LIN {X 0,Y 449.895,Z 770.969,A -85,B 0,C 180,E1 -4613.165,E2 -4613.165} C_VEL
LIN {X 0,Y 451.158,Z 755.212,A -85,B 0,C 180,E1 -4614.344,E2 -4614.344} C_VEL
LIN {X 0,Y 452.253,Z 738.74,A -85,B 0,C 180,E1 -4615.328,E2 -4615.328} C_VEL
LIN {X 0,Y 453.129,Z 720.861,A -85,B 0,C 180,E1 -4616.147,E2 -4616.147} C_VEL
LIN {X 0,Y 453.677,Z 702.427,A -85,B 0,C 180,E1 -4616.749,E2 -4616.749} C_VEL
LIN {X 0,Y 453.972,Z 680.153,A -85,B 0,C 180,E1 -4617.195,E2 -4617.195} C_VEL
LIN {X 0,Y 457.144,Z 495.027,A -85,B 0,C 180,E1 -4620.269,E2 -4620.269} C_VEL
LIN {X 0,Y 456.167,Z 488.518,A -85,B 0,C 180,E1 -4620.474,E2 -4620.474} C_VEL
LIN {X 0,Y 456.984,Z 456.622,A -85,B 0,C 180,E1 -4622.788,E2 -4622.788} C_VEL
LIN {X 0,Y 458.772,Z 418.991,A -85,B 0,C 180,E1 -4625.739,E2 -4625.739} C_VEL
LIN {X 0,Y 451.224,Z 399.096,A -85,B 0,C 180,E1 -4628.127,E2 -4628.127} C_VEL
LIN {X 0,Y 444.43,Z 383.394,A -85,B 0,C 180,E1 -4630.1,E2 -4630.1} C_VEL
LIN {X 0,Y 441.262,Z 376.238,A -85,B 0,C 180,E1 -4631.014,E2 -4631.014} C_VEL
LIN {X 0,Y 441.194,Z 375.762,A -85,B 0,C 180,E1 -4631.088,E2 -4631.088} C_VEL
LIN {X 0,Y 441.156,Z 375.762,A -85,B 0,C 180,E1 -4634.819,E2 -4634.819} C_VEL
LIN {X 0,Y 441.18,Z 375.869,A -85,B 0,C 180,E1 -4634.958,E2 -4634.958} C_VEL
LIN {X 0,Y 442.687,Z 379.535,A -85,B 0,C 180,E1 -4635.559,E2 -4635.559} C_VEL
LIN {X 0,Y 450.981,Z 398.056,A -85,B 0,C 180,E1 -4638.537,E2 -4638.537} C_VEL
LIN {X 0,Y 459.04,Z 417.845,A -85,B 0,C 180,E1 -4641.441,E2 -4641.441} C_VEL
LIN {X 0,Y 461.711,Z 425.418,A -85,B 0,C 180,E1 -4642.476,E2 -4642.476} C_VEL
LIN {X 0,Y 458.465,Z 467.127,A -85,B 0,C 180,E1 -4646.211,E2 -4646.211} C_VEL
LIN {X 0,Y 455.403,Z 509.659,A -85,B 0,C 180,E1 -4649.961,E2 -4649.961} C_VEL
LIN {X 0,Y 452.531,Z 553.564,A -85,B 0,C 180,E1 -4653.775,E2 -4653.775} C_VEL
LIN {X 0,Y 449.914,Z 598.968,A -85,B 0,C 180,E1 -4657.665,E2 -4657.665} C_VEL
LIN {X 0,Y 450.757,Z 607.685,A -85,B 0,C 180,E1 -4657.915,E2 -4657.915} C_VEL
LIN {X 0,Y 447.26,Z 745.636,A -85,B 0,C 180,E1 -4660.73,E2 -4660.73} C_VEL
LIN {X 0,Y 446.843,Z 762.879,A -85,B 0,C 180,E1 -4661.338,E2 -4661.338} C_VEL
LIN {X 0,Y 446.246,Z 778.27,A -85,B 0,C 180,E1 -4662.123,E2 -4662.123} C_VEL
LIN {X 0,Y 445.489,Z 793.673,A -85,B 0,C 180,E1 -4663.17,E2 -4663.17} C_VEL
LIN {X 0,Y 444.687,Z 807.201,A -85,B 0,C 180,E1 -4664.346,E2 -4664.346} C_VEL
LIN {X 0,Y 443.839,Z 820.409,A -85,B 0,C 180,E1 -4665.785,E2 -4665.785} C_VEL
LIN {X 0,Y 443.061,Z 831.979,A -85,B 0,C 180,E1 -4667.355,E2 -4667.355} C_VEL
LIN {X 0,Y 442.35,Z 842.758,A -85,B 0,C 180,E1 -4669.186,E2 -4669.186} C_VEL
LIN {X 0,Y 441.823,Z 851.245,A -85,B 0,C 180,E1 -4671.016,E2 -4671.016} C_VEL
LIN {X 0,Y 441.424,Z 858.712,A -85,B 0,C 180,E1 -4673.105,E2 -4673.105} C_VEL
LIN {X 0,Y 441.19,Z 863.794,A -85,B 0,C 180,E1 -4675.059,E2 -4675.059} C_VEL
LIN {X 0,Y 441.097,Z 867.62,A -85,B 0,C 180,E1 -4677.271,E2 -4677.271} C_VEL
LIN {X 0,Y 441.088,Z 869.436,A -85,B 0,C 180,E1 -4679.35,E2 -4679.35} C_VEL
LIN {X 0,Y 441.194,Z 869.55,A -85,B 0,C 180,E1 -4681.558,E2 -4681.558} C_VEL
LIN {X 0,Y 441.366,Z 867.927,A -85,B 0,C 180,E1 -4683.636,E2 -4683.636} C_VEL
LIN {X 0,Y 441.715,Z 864.344,A -85,B 0,C 180,E1 -4685.846,E2 -4685.846} C_VEL
LIN {X 0,Y 442.16,Z 859.396,A -85,B 0,C 180,E1 -4687.797,E2 -4687.797} C_VEL
LIN {X 0,Y 442.811,Z 852.654,A -85,B 0,C 180,E1 -4689.75,E2 -4689.75} C_VEL
LIN {X 0,Y 443.571,Z 844.422,A -85,B 0,C 180,E1 -4691.573,E2 -4691.573} C_VEL
LIN {X 0,Y 444.542,Z 833.949,A -85,B 0,C 180,E1 -4693.395,E2 -4693.395} C_VEL
LIN {X 0,Y 445.533,Z 822.497,A -85,B 0,C 180,E1 -4694.956,E2 -4694.956} C_VEL
LIN {X 0,Y 446.52,Z 810.059,A -85,B 0,C 180,E1 -4696.321,E2 -4696.321} C_VEL
LIN {X 0,Y 447.465,Z 795.723,A -85,B 0,C 180,E1 -4697.557,E2 -4697.557} C_VEL
LIN {X 0,Y 448.16,Z 782.092,A -85,B 0,C 180,E1 -4698.47,E2 -4698.47} C_VEL
LIN {X 0,Y 448.749,Z 765.732,A -85,B 0,C 180,E1 -4699.288,E2 -4699.288} C_VEL
LIN {X 0,Y 449.106,Z 747.084,A -85,B 0,C 180,E1 -4699.911,E2 -4699.911} C_VEL
LIN {X 0,Y 452.046,Z 696.665,A -85,B 0,C 180,E1 -4701.377,E2 -4701.377} C_VEL
LIN {X 0,Y 458.354,Z 622.755,A -85,B 0,C 180,E1 -4703.596,E2 -4703.596} C_VEL
LIN {X 0,Y 461.651,Z 613.359,A -85,B 0,C 180,E1 -4704.241,E2 -4704.241} C_VEL
LIN {X 0,Y 468.36,Z 575.653,A -85,B 0,C 180,E1 -4708.081,E2 -4708.081} C_VEL
LIN {X 0,Y 475.645,Z 546.296,A -85,B 0,C 180,E1 -4711.28,E2 -4711.28} C_VEL
LIN {X 0,Y 482.867,Z 525.512,A -85,B 0,C 180,E1 -4713.706,E2 -4713.706} C_VEL
LIN {X 0,Y 490.96,Z 508.824,A -85,B 0,C 180,E1 -4715.802,E2 -4715.802} C_VEL
LIN {X 0,Y 485.466,Z 518.576,A -85,B 0,C 180,E1 -4717.344,E2 -4717.344} C_VEL
LIN {X 0,Y 482.77,Z 527.164,A -85,B 0,C 180,E1 -4718.716,E2 -4718.716} C_VEL
LIN {X 0,Y 482.118,Z 536.127,A -85,B 0,C 180,E1 -4720.164,E2 -4720.164} C_VEL
LIN {X 0,Y 483.586,Z 544.905,A -85,B 0,C 180,E1 -4721.582,E2 -4721.582} C_VEL
LIN {X 0,Y 487.497,Z 554.414,A -85,B 0,C 180,E1 -4723.1,E2 -4723.1} C_VEL
LIN {X 0,Y 493.464,Z 563.318,A -85,B 0,C 180,E1 -4724.512,E2 -4724.512} C_VEL
LIN {X 0,Y 501.507,Z 571.927,A -85,B 0,C 180,E1 -4725.867,E2 -4725.867} C_VEL
LIN {X 0,Y 512.262,Z 580.404,A -85,B 0,C 180,E1 -4727.214,E2 -4727.214} C_VEL
LIN {X 0,Y 520.948,Z 586.006,A -85,B 0,C 180,E1 -4728.093,E2 -4728.093} C_VEL
LIN {X 0,Y 500.898,Z 618.864,A -85,B 0,C 180,E1 -4728.811,E2 -4728.811} C_VEL
LIN {X 0,Y 489.956,Z 639.653,A -85,B 0,C 180,E1 -4729.388,E2 -4729.388} C_VEL
LIN {X 0,Y 482.648,Z 656.795,A -85,B 0,C 180,E1 -4729.989,E2 -4729.989} C_VEL
LIN {X 0,Y 479.917,Z 663.519,A -85,B 0,C 180,E1 -4730.237,E2 -4730.237} C_VEL
LIN {X 0,Y 472.657,Z 680.377,A -85,B 0,C 180,E1 -4730.843,E2 -4730.843} C_VEL
LIN {X 0,Y 463.801,Z 707.381,A -85,B 0,C 180,E1 -4732.013,E2 -4732.013} C_VEL
LIN {X 0,Y 462.854,Z 711.533,A -85,B 0,C 180,E1 -4732.171,E2 -4732.171} C_VEL
LIN {X 0,Y 461.732,Z 725.369,A -85,B 0,C 180,E1 -4732.362,E2 -4732.362} C_VEL
LIN {X 0,Y 460.813,Z 757.516,A -85,B 0,C 180,E1 -4732.978,E2 -4732.978} C_VEL
LIN {X 0,Y 459.501,Z 781.218,A -85,B 0,C 180,E1 -4733.648,E2 -4733.648} C_VEL
LIN {X 0,Y 457.971,Z 803.987,A -85,B 0,C 180,E1 -4734.522,E2 -4734.522} C_VEL
LIN {X 0,Y 456.223,Z 826.917,A -85,B 0,C 180,E1 -4735.643,E2 -4735.643} C_VEL
LIN {X 0,Y 454.282,Z 849.228,A -85,B 0,C 180,E1 -4736.988,E2 -4736.988} C_VEL
LIN {X 0,Y 452.395,Z 869.681,A -85,B 0,C 180,E1 -4738.486,E2 -4738.486} C_VEL
LIN {X 0,Y 450.357,Z 889.784,A -85,B 0,C 180,E1 -4740.235,E2 -4740.235} C_VEL
LIN {X 0,Y 448.559,Z 907.091,A -85,B 0,C 180,E1 -4741.998,E2 -4741.998} C_VEL
LIN {X 0,Y 446.629,Z 925.029,A -85,B 0,C 180,E1 -4744.151,E2 -4744.151} C_VEL
LIN {X 0,Y 444.866,Z 941.503,A -85,B 0,C 180,E1 -4746.49,E2 -4746.49} C_VEL
LIN {X 0,Y 443.317,Z 956.495,A -85,B 0,C 180,E1 -4749.024,E2 -4749.024} C_VEL
LIN {X 0,Y 442.11,Z 968.957,A -85,B 0,C 180,E1 -4751.541,E2 -4751.541} C_VEL
LIN {X 0,Y 441.355,Z 977.773,A -85,B 0,C 180,E1 -4753.685,E2 -4753.685} C_VEL
LIN {X 0,Y 440.635,Z 986.687,A -85,B 0,C 180,E1 -4756.483,E2 -4756.483} C_VEL
LIN {X 0,Y 440.219,Z 993.705,A -85,B 0,C 180,E1 -4759.266,E2 -4759.266} C_VEL
LIN {X 0,Y 440.005,Z 999.024,A -85,B 0,C 180,E1 -4762.032,E2 -4762.032} C_VEL
LIN {X 0,Y 439.912,Z 1002.741,A -85,B 0,C 180,E1 -4764.783,E2 -4764.783} C_VEL
LIN {X 0,Y 439.9,Z 1004.828,A -85,B 0,C 180,E1 -4767.525,E2 -4767.525} C_VEL
LIN {X 0,Y 439.894,Z 1005.447,A -85,B 0,C 180,E1 -4770.521,E2 -4770.521} C_VEL
LIN {X 0,Y 439.906,Z 1004.417,A -85,B 0,C 180,E1 -4773.257,E2 -4773.257} C_VEL
LIN {X 0,Y 439.948,Z 1001.676,A -85,B 0,C 180,E1 -4776.131,E2 -4776.131} C_VEL
LIN {X 0,Y 440.067,Z 997.197,A -85,B 0,C 180,E1 -4779.019,E2 -4779.019} C_VEL
LIN {X 0,Y 440.339,Z 991.238,A -85,B 0,C 180,E1 -4781.792,E2 -4781.792} C_VEL
LIN {X 0,Y 440.857,Z 983.531,A -85,B 0,C 180,E1 -4784.581,E2 -4784.581} C_VEL
LIN {X 0,Y 441.556,Z 975.224,A -85,B 0,C 180,E1 -4786.984,E2 -4786.984} C_VEL
LIN {X 0,Y 442.585,Z 964.124,A -85,B 0,C 180,E1 -4789.533,E2 -4789.533} C_VEL
LIN {X 0,Y 443.881,Z 951.647,A -85,B 0,C 180,E1 -4791.957,E2 -4791.957} C_VEL
LIN {X 0,Y 445.543,Z 936.945,A -85,B 0,C 180,E1 -4794.388,E2 -4794.388} C_VEL
LIN {X 0,Y 447.541,Z 920.085,A -85,B 0,C 180,E1 -4796.755,E2 -4796.755} C_VEL
LIN {X 0,Y 449.799,Z 901.306,A -85,B 0,C 180,E1 -4798.985,E2 -4798.985} C_VEL
LIN {X 0,Y 452.216,Z 881.067,A -85,B 0,C 180,E1 -4801.008,E2 -4801.008} C_VEL
LIN {X 0,Y 454.533,Z 861.152,A -85,B 0,C 180,E1 -4802.686,E2 -4802.686} C_VEL
LIN {X 0,Y 456.76,Z 840.526,A -85,B 0,C 180,E1 -4804.132,E2 -4804.132} C_VEL
LIN {X 0,Y 458.846,Z 819.523,A -85,B 0,C 180,E1 -4805.348,E2 -4805.348} C_VEL
LIN {X 0,Y 460.789,Z 797.618,A -85,B 0,C 180,E1 -4806.368,E2 -4806.368} C_VEL
LIN {X 0,Y 462.401,Z 775.254,A -85,B 0,C 180,E1 -4807.157,E2 -4807.157} C_VEL
LIN {X 0,Y 463.714,Z 752.034,A -85,B 0,C 180,E1 -4807.736,E2 -4807.736} C_VEL
LIN {X 0,Y 464.958,Z 716.912,A -85,B 0,C 180,E1 -4808.352,E2 -4808.352} C_VEL
LIN {X 0,Y 465.536,Z 714.104,A -85,B 0,C 180,E1 -4808.446,E2 -4808.446} C_VEL
LIN {X 0,Y 470.715,Z 697.809,A -85,B 0,C 180,E1 -4809.192,E2 -4809.192} C_VEL
LIN {X 0,Y 477.201,Z 679.573,A -85,B 0,C 180,E1 -4809.955,E2 -4809.955} C_VEL
LIN {X 0,Y 485.1,Z 661.285,A -85,B 0,C 180,E1 -4810.563,E2 -4810.563} C_VEL
LIN {X 0,Y 492.217,Z 644.342,A -85,B 0,C 180,E1 -4811.159,E2 -4811.159} C_VEL
LIN {X 0,Y 502.709,Z 623.858,A -85,B 0,C 180,E1 -4811.705,E2 -4811.705} C_VEL
LIN {X 0,Y 519.668,Z 594.789,A -85,B 0,C 180,E1 -4812.256,E2 -4812.256} C_VEL
LIN {X 0,Y 523.657,Z 588.098,A -85,B 0,C 180,E1 -4812.36,E2 -4812.36} C_VEL
LIN {X 0,Y 513.143,Z 581.511,A -85,B 0,C 180,E1 -4813.707,E2 -4813.707} C_VEL
LIN {X 0,Y 503.509,Z 573.197,A -85,B 0,C 180,E1 -4815.175,E2 -4815.175} C_VEL
LIN {X 0,Y 495.035,Z 562.874,A -85,B 0,C 180,E1 -4816.788,E2 -4816.788} C_VEL
LIN {X 0,Y 488.639,Z 551.749,A -85,B 0,C 180,E1 -4818.319,E2 -4818.319} C_VEL
LIN {X 0,Y 483.581,Z 538.76,A -85,B 0,C 180,E1 -4819.908,E2 -4819.908} C_VEL
LIN {X 0,Y 480.199,Z 523.859,A -85,B 0,C 180,E1 -4821.526,E2 -4821.526} C_VEL
LIN {X 0,Y 478.615,Z 506.943,A -85,B 0,C 180,E1 -4823.162,E2 -4823.162} C_VEL
LIN {X 0,Y 478.809,Z 488.569,A -85,B 0,C 180,E1 -4824.735,E2 -4824.735} C_VEL
LIN {X 0,Y 482.727,Z 450.056,A -85,B 0,C 180,E1 -4827.698,E2 -4827.698} C_VEL
LIN {X 0,Y 473.244,Z 432.509,A -85,B 0,C 180,E1 -4830.788,E2 -4830.788} C_VEL
LIN {X 0,Y 465.807,Z 419.157,A -85,B 0,C 180,E1 -4833.345,E2 -4833.345} C_VEL
LIN {X 0,Y 458.025,Z 405.408,A -85,B 0,C 180,E1 -4836.181,E2 -4836.181} C_VEL
LIN {X 0,Y 452.378,Z 395.654,A -85,B 0,C 180,E1 -4838.34,E2 -4838.34} C_VEL
LIN {X 0,Y 449.617,Z 390.88,A -85,B 0,C 180,E1 -4839.43,E2 -4839.43} C_VEL
LIN {X 0,Y 447.276,Z 386.724,A -85,B 0,C 180,E1 -4840.409,E2 -4840.409} C_VEL
LIN {X 0,Y 444.491,Z 382.323,A -85,B 0,C 180,E1 -4841.508,E2 -4841.508} C_VEL
LIN {X 0,Y 443.697,Z 380.667,A -85,B 0,C 180,E1 -4841.882,E2 -4841.882} C_VEL
LIN {X 0,Y 441.581,Z 377.455,A -85,B 0,C 180,E1 -4842.746,E2 -4842.746} C_VEL
LIN {X 0,Y 441.179,Z 375.776,A -85,B 0,C 180,E1 -4843.069,E2 -4843.069} C_VEL
LIN {X 0,Y 441.195,Z 375.776,A -85,B 0,C 180,E1 -4846.769,E2 -4846.769} C_VEL
LIN {X 0,Y 441.198,Z 375.777,A -85,B 0,C 180,E1 -4850.609,E2 -4850.609} C_VEL
LIN {X 0,Y 441.162,Z 375.78,A -85,B 0,C 180,E1 -4854.277,E2 -4854.277} C_VEL
LIN {X 0,Y 441.188,Z 375.781,A -85,B 0,C 180,E1 -4858.064,E2 -4858.064} C_VEL
LIN {X 0,Y 441.172,Z 375.788,A -85,B 0,C 180,E1 -4861.689,E2 -4861.689} C_VEL
LIN {X 0,Y 441.183,Z 375.78,A -85,B 0,C 180,E1 -4865.593,E2 -4865.593} C_VEL
LIN {X 0,Y 441.19,Z 375.784,A -85,B 0,C 180,E1 -4869.26,E2 -4869.26} C_VEL
LIN {X 0,Y 441.199,Z 375.777,A -85,B 0,C 180,E1 -4873.099,E2 -4873.099} C_VEL
LIN {X 0,Y 441.156,Z 375.783,A -85,B 0,C 180,E1 -4876.865,E2 -4876.865} C_VEL
LIN {X 0,Y 441.187,Z 375.777,A -85,B 0,C 180,E1 -4880.704,E2 -4880.704} C_VEL
LIN {X 0,Y 441.176,Z 375.779,A -85,B 0,C 180,E1 -4884.361,E2 -4884.361} C_VEL
LIN {X 0,Y 441.19,Z 375.774,A -85,B 0,C 180,E1 -4888.167,E2 -4888.167} C_VEL
LIN {X 0,Y 441.177,Z 375.772,A -85,B 0,C 180,E1 -4891.802,E2 -4891.802} C_VEL
LIN {X 0,Y 441.188,Z 375.75,A -85,B 0,C 180,E1 -4895.552,E2 -4895.552} C_VEL
LIN {X 0,Y 441.162,Z 375.784,A -85,B 0,C 180,E1 -4899.223,E2 -4899.223} C_VEL
LIN {X 0,Y 441.176,Z 375.758,A -85,B 0,C 180,E1 -4903.192,E2 -4903.192} C_VEL
LIN {X 0,Y 441.188,Z 375.759,A -85,B 0,C 180,E1 -4906.866,E2 -4906.866} C_VEL
LIN {X 0,Y 441.178,Z 375.864,A -85,B 0,C 180,E1 -4909.05,E2 -4909.05} C_VEL
LIN {X 0,Y 442.319,Z 379.044,A -85,B 0,C 180,E1 -4909.423,E2 -4909.423} C_VEL
LIN {X 0,Y 449.225,Z 394.2,A -85,B 0,C 180,E1 -4911.374,E2 -4911.374} C_VEL
LIN {X 0,Y 457.31,Z 415.015,A -85,B 0,C 180,E1 -4913.889,E2 -4913.889} C_VEL
LIN {X 0,Y 458.713,Z 419.428,A -85,B 0,C 180,E1 -4914.394,E2 -4914.394} C_VEL
LIN {X 0,Y 456.717,Z 463.963,A -85,B 0,C 180,E1 -4917.861,E2 -4917.861} C_VEL
LIN {X 0,Y 456.193,Z 489.039,A -85,B 0,C 180,E1 -4919.645,E2 -4919.645} C_VEL
LIN {X 0,Y 457.27,Z 497.519,A -85,B 0,C 180,E1 -4919.88,E2 -4919.88} C_VEL
LIN {X 0,Y 455.728,Z 579.645,A -85,B 0,C 180,E1 -4921.239,E2 -4921.239} C_VEL
LIN {X 0,Y 454.731,Z 587.33,A -85,B 0,C 180,E1 -4921.304,E2 -4921.304} C_VEL
LIN {X 0,Y 448.905,Z 607.766,A -85,B 0,C 180,E1 -4921.25,E2 -4921.25} C_VEL
LIN {X 0,Y 448.139,Z 614.363,A -85,B 0,C 180,E1 -4921.313,E2 -4921.313} C_VEL
LIN {X 0,Y 446.692,Z 698.387,A -85,B 0,C 180,E1 -4922.759,E2 -4922.759} C_VEL
LIN {X 0,Y 446.206,Z 717.049,A -85,B 0,C 180,E1 -4923.307,E2 -4923.307} C_VEL
LIN {X 0,Y 445.434,Z 734.356,A -85,B 0,C 180,E1 -4924.042,E2 -4924.042} C_VEL
LIN {X 0,Y 444.36,Z 751.044,A -85,B 0,C 180,E1 -4924.975,E2 -4924.975} C_VEL
LIN {X 0,Y 443.083,Z 767.04,A -85,B 0,C 180,E1 -4926.106,E2 -4926.106} C_VEL
LIN {X 0,Y 441.617,Z 782.989,A -85,B 0,C 180,E1 -4927.504,E2 -4927.504} C_VEL
LIN {X 0,Y 440.106,Z 797.217,A -85,B 0,C 180,E1 -4929.026,E2 -4929.026} C_VEL
LIN {X 0,Y 438.635,Z 810.198,A -85,B 0,C 180,E1 -4930.7,E2 -4930.7} C_VEL
LIN {X 0,Y 437.22,Z 822.243,A -85,B 0,C 180,E1 -4932.568,E2 -4932.568} C_VEL
LIN {X 0,Y 435.957,Z 832.923,A -85,B 0,C 180,E1 -4934.571,E2 -4934.571} C_VEL
LIN {X 0,Y 434.91,Z 842.254,A -85,B 0,C 180,E1 -4936.709,E2 -4936.709} C_VEL
LIN {X 0,Y 434.07,Z 850.212,A -85,B 0,C 180,E1 -4938.978,E2 -4938.978} C_VEL
LIN {X 0,Y 433.464,Z 856.74,A -85,B 0,C 180,E1 -4941.377,E2 -4941.377} C_VEL
LIN {X 0,Y 433.089,Z 861.745,A -85,B 0,C 180,E1 -4943.904,E2 -4943.904} C_VEL
LIN {X 0,Y 432.882,Z 864.947,A -85,B 0,C 180,E1 -4946.425,E2 -4946.425} C_VEL
LIN {X 0,Y 432.788,Z 866.472,A -85,B 0,C 180,E1 -4948.941,E2 -4948.941} C_VEL
LIN {X 0,Y 432.796,Z 866.367,A -85,B 0,C 180,E1 -4951.457,E2 -4951.457} C_VEL
LIN {X 0,Y 432.903,Z 864.627,A -85,B 0,C 180,E1 -4953.974,E2 -4953.974} C_VEL
LIN {X 0,Y 433.119,Z 861.2,A -85,B 0,C 180,E1 -4956.495,E2 -4956.495} C_VEL
LIN {X 0,Y 433.497,Z 856.304,A -85,B 0,C 180,E1 -4958.89,E2 -4958.89} C_VEL
LIN {X 0,Y 434.125,Z 849.646,A -85,B 0,C 180,E1 -4961.29,E2 -4961.29} C_VEL
LIN {X 0,Y 435.045,Z 841.005,A -85,B 0,C 180,E1 -4963.694,E2 -4963.694} C_VEL
LIN {X 0,Y 436.135,Z 831.387,A -85,B 0,C 180,E1 -4965.832,E2 -4965.832} C_VEL
LIN {X 0,Y 437.446,Z 820.381,A -85,B 0,C 180,E1 -4967.836,E2 -4967.836} C_VEL
LIN {X 0,Y 438.9,Z 807.956,A -85,B 0,C 180,E1 -4969.704,E2 -4969.704} C_VEL
LIN {X 0,Y 440.469,Z 794.007,A -85,B 0,C 180,E1 -4971.437,E2 -4971.437} C_VEL
LIN {X 0,Y 441.948,Z 779.713,A -85,B 0,C 180,E1 -4972.901,E2 -4972.901} C_VEL
LIN {X 0,Y 443.361,Z 763.881,A -85,B 0,C 180,E1 -4974.233,E2 -4974.233} C_VEL
LIN {X 0,Y 444.662,Z 747.183,A -85,B 0,C 180,E1 -4975.356,E2 -4975.356} C_VEL
LIN {X 0,Y 445.68,Z 729.87,A -85,B 0,C 180,E1 -4976.265,E2 -4976.265} C_VEL
LIN {X 0,Y 446.429,Z 711.294,A -85,B 0,C 180,E1 -4976.984,E2 -4976.984} C_VEL
LIN {X 0,Y 446.792,Z 692.057,A -85,B 0,C 180,E1 -4977.472,E2 -4977.472} C_VEL
LIN {X 0,Y 450.296,Z 496.276,A -85,B 0,C 180,E1 -4980.775,E2 -4980.775} C_VEL
LIN {X 0,Y 449.33,Z 489.417,A -85,B 0,C 180,E1 -4981.007,E2 -4981.007} C_VEL
LIN {X 0,Y 450.226,Z 456.889,A -85,B 0,C 180,E1 -4983.382,E2 -4983.382} C_VEL
LIN {X 0,Y 451.856,Z 422.041,A -85,B 0,C 180,E1 -4986.131,E2 -4986.131} C_VEL
LIN {X 0,Y 444.344,Z 402.144,A -85,B 0,C 180,E1 -4988.558,E2 -4988.558} C_VEL
LIN {X 0,Y 436.424,Z 384.18,A -85,B 0,C 180,E1 -4990.883,E2 -4990.883} C_VEL
LIN {X 0,Y 433.275,Z 377.154,A -85,B 0,C 180,E1 -4991.808,E2 -4991.808} C_VEL
LIN {X 0,Y 433.212,Z 376.766,A -85,B 0,C 180,E1 -4991.913,E2 -4991.913} C_VEL
LIN {X 0,Y 433.233,Z 376.945,A -85,B 0,C 180,E1 -4994.04,E2 -4994.04} C_VEL
LIN {X 0,Y 434.493,Z 380.206,A -85,B 0,C 180,E1 -4994.578,E2 -4994.578} C_VEL
LIN {X 0,Y 440.848,Z 393.997,A -85,B 0,C 180,E1 -4996.913,E2 -4996.913} C_VEL
LIN {X 0,Y 448.471,Z 411.79,A -85,B 0,C 180,E1 -4999.684,E2 -4999.684} C_VEL
LIN {X 0,Y 454.942,Z 428.636,A -85,B 0,C 180,E1 -5002.093,E2 -5002.093} C_VEL
LIN {X 0,Y 451.513,Z 470.101,A -85,B 0,C 180,E1 -5005.849,E2 -5005.849} C_VEL
LIN {X 0,Y 448.254,Z 513.147,A -85,B 0,C 180,E1 -5009.682,E2 -5009.682} C_VEL
LIN {X 0,Y 445.243,Z 556.959,A -85,B 0,C 180,E1 -5013.528,E2 -5013.528} C_VEL
LIN {X 0,Y 442.695,Z 600.382,A -85,B 0,C 180,E1 -5017.26,E2 -5017.26} C_VEL
LIN {X 0,Y 443.485,Z 608.695,A -85,B 0,C 180,E1 -5017.498,E2 -5017.498} C_VEL
LIN {X 0,Y 439.729,Z 746.682,A -85,B 0,C 180,E1 -5020.399,E2 -5020.399} C_VEL
LIN {X 0,Y 439.297,Z 763.537,A -85,B 0,C 180,E1 -5021.005,E2 -5021.005} C_VEL
LIN {X 0,Y 438.673,Z 779.026,A -85,B 0,C 180,E1 -5021.804,E2 -5021.804} C_VEL
LIN {X 0,Y 437.875,Z 794.478,A -85,B 0,C 180,E1 -5022.868,E2 -5022.868} C_VEL
LIN {X 0,Y 437.034,Z 808.084,A -85,B 0,C 180,E1 -5024.065,E2 -5024.065} C_VEL
LIN {X 0,Y 436.105,Z 821.82,A -85,B 0,C 180,E1 -5025.587,E2 -5025.587} C_VEL
LIN {X 0,Y 435.314,Z 832.983,A -85,B 0,C 180,E1 -5027.126,E2 -5027.126} C_VEL
LIN {X 0,Y 434.556,Z 843.815,A -85,B 0,C 180,E1 -5028.99,E2 -5028.99} C_VEL
LIN {X 0,Y 433.994,Z 852.372,A -85,B 0,C 180,E1 -5030.853,E2 -5030.853} C_VEL
LIN {X 0,Y 433.564,Z 859.891,A -85,B 0,C 180,E1 -5032.979,E2 -5032.979} C_VEL
LIN {X 0,Y 433.315,Z 865.041,A -85,B 0,C 180,E1 -5034.969,E2 -5034.969} C_VEL
LIN {X 0,Y 433.211,Z 868.921,A -85,B 0,C 180,E1 -5037.222,E2 -5037.222} C_VEL
LIN {X 0,Y 433.206,Z 870.802,A -85,B 0,C 180,E1 -5039.338,E2 -5039.338} C_VEL
LIN {X 0,Y 433.324,Z 870.975,A -85,B 0,C 180,E1 -5041.586,E2 -5041.586} C_VEL
LIN {X 0,Y 433.519,Z 869.405,A -85,B 0,C 180,E1 -5043.702,E2 -5043.702} C_VEL
LIN {X 0,Y 433.903,Z 865.878,A -85,B 0,C 180,E1 -5045.952,E2 -5045.952} C_VEL
LIN {X 0,Y 434.432,Z 860.604,A -85,B 0,C 180,E1 -5048.07,E2 -5048.07} C_VEL
LIN {X 0,Y 435.162,Z 853.836,A -85,B 0,C 180,E1 -5050.056,E2 -5050.056} C_VEL
LIN {X 0,Y 435.992,Z 845.507,A -85,B 0,C 180,E1 -5051.911,E2 -5051.911} C_VEL
LIN {X 0,Y 436.97,Z 835.794,A -85,B 0,C 180,E1 -5053.631,E2 -5053.631} C_VEL
LIN {X 0,Y 438.035,Z 824.492,A -85,B 0,C 180,E1 -5055.218,E2 -5055.218} C_VEL
LIN {X 0,Y 439.094,Z 812.235,A -85,B 0,C 180,E1 -5056.605,E2 -5056.605} C_VEL
LIN {X 0,Y 440.162,Z 797.32,A -85,B 0,C 180,E1 -5057.926,E2 -5057.926} C_VEL
LIN {X 0,Y 440.907,Z 783.789,A -85,B 0,C 180,E1 -5058.853,E2 -5058.853} C_VEL
LIN {X 0,Y 441.547,Z 767.692,A -85,B 0,C 180,E1 -5059.684,E2 -5059.684} C_VEL
LIN {X 0,Y 442.067,Z 746.157,A -85,B 0,C 180,E1 -5060.427,E2 -5060.427} C_VEL
LIN {X 0,Y 445.992,Z 690.299,A -85,B 0,C 180,E1 -5062.164,E2 -5062.164} C_VEL
LIN {X 0,Y 451.973,Z 626.185,A -85,B 0,C 180,E1 -5064.158,E2 -5064.158} C_VEL
LIN {X 0,Y 455.898,Z 615.345,A -85,B 0,C 180,E1 -5064.903,E2 -5064.903} C_VEL
LIN {X 0,Y 462.809,Z 579.928,A -85,B 0,C 180,E1 -5068.589,E2 -5068.589} C_VEL
LIN {X 0,Y 470.333,Z 552.205,A -85,B 0,C 180,E1 -5071.674,E2 -5071.674} C_VEL
LIN {X 0,Y 478.011,Z 531.913,A -85,B 0,C 180,E1 -5074.095,E2 -5074.095} C_VEL
LIN {X 0,Y 484.975,Z 518.297,A -85,B 0,C 180,E1 -5075.88,E2 -5075.88} C_VEL
LIN {X 0,Y 480.047,Z 527.435,A -85,B 0,C 180,E1 -5077.382,E2 -5077.382} C_VEL
LIN {X 0,Y 477.6,Z 536.105,A -85,B 0,C 180,E1 -5078.85,E2 -5078.85} C_VEL
LIN {X 0,Y 477.346,Z 544.72,A -85,B 0,C 180,E1 -5080.319,E2 -5080.319} C_VEL
LIN {X 0,Y 479.119,Z 553.071,A -85,B 0,C 180,E1 -5081.736,E2 -5081.736} C_VEL
LIN {X 0,Y 483.287,Z 562.227,A -85,B 0,C 180,E1 -5083.26,E2 -5083.26} C_VEL
LIN {X 0,Y 489.877,Z 571.351,A -85,B 0,C 180,E1 -5084.761,E2 -5084.761} C_VEL
LIN {X 0,Y 498.107,Z 579.598,A -85,B 0,C 180,E1 -5086.106,E2 -5086.106} C_VEL
LIN {X 0,Y 508.993,Z 587.809,A -85,B 0,C 180,E1 -5087.446,E2 -5087.446} C_VEL
LIN {X 0,Y 511.176,Z 589.511,A -85,B 0,C 180,E1 -5087.693,E2 -5087.693} C_VEL
LIN {X 0,Y 493.865,Z 618.299,A -85,B 0,C 180,E1 -5088.312,E2 -5088.312} C_VEL
LIN {X 0,Y 483.367,Z 638.443,A -85,B 0,C 180,E1 -5088.868,E2 -5088.868} C_VEL
LIN {X 0,Y 475.936,Z 655.882,A -85,B 0,C 180,E1 -5089.48,E2 -5089.48} C_VEL
LIN {X 0,Y 473.072,Z 662.724,A -85,B 0,C 180,E1 -5089.728,E2 -5089.728} C_VEL
LIN {X 0,Y 465.94,Z 679.367,A -85,B 0,C 180,E1 -5090.327,E2 -5090.327} C_VEL
LIN {X 0,Y 456.689,Z 707.38,A -85,B 0,C 180,E1 -5091.553,E2 -5091.553} C_VEL
LIN {X 0,Y 456.112,Z 710.578,A -85,B 0,C 180,E1 -5091.643,E2 -5091.643} C_VEL
LIN {X 0,Y 454.845,Z 725.175,A -85,B 0,C 180,E1 -5091.848,E2 -5091.848} C_VEL
LIN {X 0,Y 453.817,Z 756.663,A -85,B 0,C 180,E1 -5092.479,E2 -5092.479} C_VEL
LIN {X 0,Y 452.315,Z 780.992,A -85,B 0,C 180,E1 -5093.197,E2 -5093.197} C_VEL
LIN {X 0,Y 450.539,Z 805.281,A -85,B 0,C 180,E1 -5094.169,E2 -5094.169} C_VEL
LIN {X 0,Y 448.706,Z 827.687,A -85,B 0,C 180,E1 -5095.31,E2 -5095.31} C_VEL
LIN {X 0,Y 446.682,Z 849.303,A -85,B 0,C 180,E1 -5096.665,E2 -5096.665} C_VEL
LIN {X 0,Y 444.565,Z 871.019,A -85,B 0,C 180,E1 -5098.306,E2 -5098.306} C_VEL
LIN {X 0,Y 442.52,Z 890.418,A -85,B 0,C 180,E1 -5100.043,E2 -5100.043} C_VEL
LIN {X 0,Y 440.595,Z 908.079,A -85,B 0,C 180,E1 -5101.908,E2 -5101.908} C_VEL
LIN {X 0,Y 438.787,Z 924.352,A -85,B 0,C 180,E1 -5103.909,E2 -5103.909} C_VEL
LIN {X 0,Y 436.997,Z 940.598,A -85,B 0,C 180,E1 -5106.253,E2 -5106.253} C_VEL
LIN {X 0,Y 435.422,Z 955.425,A -85,B 0,C 180,E1 -5108.795,E2 -5108.795} C_VEL
LIN {X 0,Y 434.138,Z 968.434,A -85,B 0,C 180,E1 -5111.468,E2 -5111.468} C_VEL
LIN {X 0,Y 433.197,Z 979.369,A -85,B 0,C 180,E1 -5114.195,E2 -5114.195} C_VEL
LIN {X 0,Y 432.581,Z 987.828,A -85,B 0,C 180,E1 -5116.772,E2 -5116.772} C_VEL
LIN {X 0,Y 432.22,Z 994.296,A -85,B 0,C 180,E1 -5119.335,E2 -5119.335} C_VEL
LIN {X 0,Y 431.995,Z 999.442,A -85,B 0,C 180,E1 -5122.151,E2 -5122.151} C_VEL
LIN {X 0,Y 431.912,Z 1002.872,A -85,B 0,C 180,E1 -5124.82,E2 -5124.82} C_VEL
LIN {X 0,Y 431.907,Z 1005.059,A -85,B 0,C 180,E1 -5127.877,E2 -5127.877} C_VEL
LIN {X 0,Y 431.901,Z 1005.406,A -85,B 0,C 180,E1 -5130.928,E2 -5130.928} C_VEL
LIN {X 0,Y 431.914,Z 1004.126,A -85,B 0,C 180,E1 -5133.716,E2 -5133.716} C_VEL
LIN {X 0,Y 431.961,Z 1001.343,A -85,B 0,C 180,E1 -5136.512,E2 -5136.512} C_VEL
LIN {X 0,Y 432.101,Z 996.72,A -85,B 0,C 180,E1 -5139.456,E2 -5139.456} C_VEL
LIN {X 0,Y 432.375,Z 991.145,A -85,B 0,C 180,E1 -5142.012,E2 -5142.012} C_VEL
LIN {X 0,Y 432.887,Z 983.264,A -85,B 0,C 180,E1 -5144.718,E2 -5144.718} C_VEL
LIN {X 0,Y 433.759,Z 972.897,A -85,B 0,C 180,E1 -5147.576,E2 -5147.576} C_VEL
LIN {X 0,Y 434.955,Z 960.837,A -85,B 0,C 180,E1 -5150.31,E2 -5150.31} C_VEL
LIN {X 0,Y 436.566,Z 946.347,A -85,B 0,C 180,E1 -5153.056,E2 -5153.056} C_VEL
LIN {X 0,Y 438.492,Z 930.371,A -85,B 0,C 180,E1 -5155.601,E2 -5155.601} C_VEL
LIN {X 0,Y 440.683,Z 912.921,A -85,B 0,C 180,E1 -5157.952,E2 -5157.952} C_VEL
LIN {X 0,Y 443.1,Z 894.048,A -85,B 0,C 180,E1 -5160.105,E2 -5160.105} C_VEL
LIN {X 0,Y 445.545,Z 874.584,A -85,B 0,C 180,E1 -5161.979,E2 -5161.979} C_VEL
LIN {X 0,Y 447.972,Z 854.051,A -85,B 0,C 180,E1 -5163.642,E2 -5163.642} C_VEL
LIN {X 0,Y 450.32,Z 833.716,A -85,B 0,C 180,E1 -5165.018,E2 -5165.018} C_VEL
LIN {X 0,Y 452.409,Z 813.009,A -85,B 0,C 180,E1 -5166.163,E2 -5166.163} C_VEL
LIN {X 0,Y 454.376,Z 790.662,A -85,B 0,C 180,E1 -5167.145,E2 -5167.145} C_VEL
LIN {X 0,Y 456.081,Z 768.238,A -85,B 0,C 180,E1 -5167.885,E2 -5167.885} C_VEL
LIN {X 0,Y 457.24,Z 745.376,A -85,B 0,C 180,E1 -5168.411,E2 -5168.411} C_VEL
LIN {X 0,Y 458.338,Z 716.737,A -85,B 0,C 180,E1 -5168.91,E2 -5168.91} C_VEL
LIN {X 0,Y 458.707,Z 714.271,A -85,B 0,C 180,E1 -5168.965,E2 -5168.965} C_VEL
LIN {X 0,Y 463.894,Z 697.959,A -85,B 0,C 180,E1 -5169.722,E2 -5169.722} C_VEL
LIN {X 0,Y 471.193,Z 677.872,A -85,B 0,C 180,E1 -5170.566,E2 -5170.566} C_VEL
LIN {X 0,Y 478.75,Z 660.7,A -85,B 0,C 180,E1 -5171.137,E2 -5171.137} C_VEL
LIN {X 0,Y 485.877,Z 643.747,A -85,B 0,C 180,E1 -5171.737,E2 -5171.737} C_VEL
LIN {X 0,Y 496.338,Z 623.24,A -85,B 0,C 180,E1 -5172.286,E2 -5172.286} C_VEL
LIN {X 0,Y 512.519,Z 595.512,A -85,B 0,C 180,E1 -5172.818,E2 -5172.818} C_VEL
LIN {X 0,Y 514.44,Z 592.027,A -85,B 0,C 180,E1 -5172.885,E2 -5172.885} C_VEL
LIN {X 0,Y 503.066,Z 583.705,A -85,B 0,C 180,E1 -5174.478,E2 -5174.478} C_VEL
LIN {X 0,Y 493.966,Z 574.401,A -85,B 0,C 180,E1 -5176.03,E2 -5176.03} C_VEL
LIN {X 0,Y 486.464,Z 563.794,A -85,B 0,C 180,E1 -5177.612,E2 -5177.612} C_VEL
LIN {X 0,Y 480.141,Z 550.777,A -85,B 0,C 180,E1 -5179.323,E2 -5179.323} C_VEL
LIN {X 0,Y 475.888,Z 537.088,A -85,B 0,C 180,E1 -5180.927,E2 -5180.927} C_VEL
LIN {X 0,Y 473.336,Z 521.87,A -85,B 0,C 180,E1 -5182.529,E2 -5182.529} C_VEL
LIN {X 0,Y 472.382,Z 504.471,A -85,B 0,C 180,E1 -5184.161,E2 -5184.161} C_VEL
LIN {X 0,Y 473.345,Z 484.704,A -85,B 0,C 180,E1 -5185.815,E2 -5185.815} C_VEL
LIN {X 0,Y 476.696,Z 454.363,A -85,B 0,C 180,E1 -5188.154,E2 -5188.154} C_VEL
LIN {X 0,Y 466.421,Z 435.205,A -85,B 0,C 180,E1 -5191.583,E2 -5191.583} C_VEL
LIN {X 0,Y 458.357,Z 420.846,A -85,B 0,C 180,E1 -5194.411,E2 -5194.411} C_VEL
LIN {X 0,Y 450.377,Z 406.754,A -85,B 0,C 180,E1 -5197.414,E2 -5197.414} C_VEL
LIN {X 0,Y 444.477,Z 396.71,A -85,B 0,C 180,E1 -5199.732,E2 -5199.732} C_VEL
LIN {X 0,Y 441.442,Z 391.577,A -85,B 0,C 180,E1 -5200.965,E2 -5200.965} C_VEL
LIN {X 0,Y 438.544,Z 386.541,A -85,B 0,C 180,E1 -5202.211,E2 -5202.211} C_VEL
LIN {X 0,Y 436.499,Z 383.05,A -85,B 0,C 180,E1 -5203.088,E2 -5203.088} C_VEL
LIN {X 0,Y 436.016,Z 381.883,A -85,B 0,C 180,E1 -5203.343,E2 -5203.343} C_VEL
LIN {X 0,Y 433.833,Z 378.903,A -85,B 0,C 180,E1 -5204.22,E2 -5204.22} C_VEL
LIN {X 0,Y 433.26,Z 376.762,A -85,B 0,C 180,E1 -5204.686,E2 -5204.686} C_VEL
LIN {X 0,Y 433.244,Z 376.766,A -85,B 0,C 180,E1 -5208.418,E2 -5208.418} C_VEL
LIN {X 0,Y 433.247,Z 376.766,A -85,B 0,C 180,E1 -5212.175,E2 -5212.175} C_VEL
LIN {X 0,Y 433.217,Z 376.772,A -85,B 0,C 180,E1 -5216.03,E2 -5216.03} C_VEL
LIN {X 0,Y 433.262,Z 376.773,A -85,B 0,C 180,E1 -5219.736,E2 -5219.736} C_VEL
LIN {X 0,Y 433.223,Z 376.776,A -85,B 0,C 180,E1 -5223.573,E2 -5223.573} C_VEL
LIN {X 0,Y 433.265,Z 376.769,A -85,B 0,C 180,E1 -5227.292,E2 -5227.292} C_VEL
LIN {X 0,Y 433.247,Z 376.771,A -85,B 0,C 180,E1 -5231.178,E2 -5231.178} C_VEL
LIN {X 0,Y 433.245,Z 376.766,A -85,B 0,C 180,E1 -5234.843,E2 -5234.843} C_VEL
LIN {X 0,Y 433.216,Z 376.769,A -85,B 0,C 180,E1 -5238.712,E2 -5238.712} C_VEL
LIN {X 0,Y 433.262,Z 376.768,A -85,B 0,C 180,E1 -5242.382,E2 -5242.382} C_VEL
LIN {X 0,Y 433.233,Z 376.766,A -85,B 0,C 180,E1 -5246.156,E2 -5246.156} C_VEL
LIN {X 0,Y 433.257,Z 376.766,A -85,B 0,C 180,E1 -5249.806,E2 -5249.806} C_VEL
LIN {X 0,Y 433.233,Z 376.771,A -85,B 0,C 180,E1 -5253.635,E2 -5253.635} C_VEL
LIN {X 0,Y 433.245,Z 376.735,A -85,B 0,C 180,E1 -5257.371,E2 -5257.371} C_VEL
LIN {X 0,Y 433.209,Z 376.754,A -85,B 0,C 180,E1 -5261.2,E2 -5261.2} C_VEL
LIN {X 0,Y 433.258,Z 376.772,A -85,B 0,C 180,E1 -5264.925,E2 -5264.925} C_VEL
LIN {X 0,Y 433.235,Z 376.77,A -85,B 0,C 180,E1 -5268.261,E2 -5268.261} C_VEL
LIN {X 0,Y 434.46,Z 380.101,A -85,B 0,C 180,E1 -5268.663,E2 -5268.663} C_VEL
LIN {X 0,Y 441.669,Z 395.755,A -85,B 0,C 180,E1 -5270.735,E2 -5270.735} C_VEL
LIN {X 0,Y 449.512,Z 415.674,A -85,B 0,C 180,E1 -5273.203,E2 -5273.203} C_VEL
LIN {X 0,Y 451.847,Z 422.595,A -85,B 0,C 180,E1 -5274.02,E2 -5274.02} C_VEL
LIN {X 0,Y 449.857,Z 466.783,A -85,B 0,C 180,E1 -5277.461,E2 -5277.461} C_VEL
LIN {X 0,Y 449.364,Z 490.343,A -85,B 0,C 180,E1 -5279.136,E2 -5279.136} C_VEL
LIN {X 0,Y 450.408,Z 498.794,A -85,B 0,C 180,E1 -5279.374,E2 -5279.374} C_VEL
LIN {X 0,Y 448.139,Z 614.363,A -85,B 0,C 180,E1 -5281.313,E2 -5281.313} C_VEL
LIN {X 0,Y 447.134,Z 622.047,A -85,B 0,C 180,E1 -5281.379,E2 -5281.379} C_VEL
LIN {X 0,Y 441.265,Z 642.471,A -85,B 0,C 180,E1 -5281.322,E2 -5281.322} C_VEL
LIN {X 0,Y 440.496,Z 649.066,A -85,B 0,C 180,E1 -5281.386,E2 -5281.386} C_VEL
LIN {X 0,Y 439.64,Z 700.343,A -85,B 0,C 180,E1 -5282.303,E2 -5282.303} C_VEL
LIN {X 0,Y 439.125,Z 718.924,A -85,B 0,C 180,E1 -5282.867,E2 -5282.867} C_VEL
LIN {X 0,Y 438.282,Z 736.634,A -85,B 0,C 180,E1 -5283.641,E2 -5283.641} C_VEL
LIN {X 0,Y 437.057,Z 754.435,A -85,B 0,C 180,E1 -5284.672,E2 -5284.672} C_VEL
LIN {X 0,Y 435.648,Z 770.859,A -85,B 0,C 180,E1 -5285.888,E2 -5285.888} C_VEL
LIN {X 0,Y 434.045,Z 786.972,A -85,B 0,C 180,E1 -5287.375,E2 -5287.375} C_VEL
LIN {X 0,Y 432.403,Z 801.343,A -85,B 0,C 180,E1 -5288.998,E2 -5288.998} C_VEL
LIN {X 0,Y 430.746,Z 814.937,A -85,B 0,C 180,E1 -5290.864,E2 -5290.864} C_VEL
LIN {X 0,Y 429.282,Z 826.561,A -85,B 0,C 180,E1 -5292.795,E2 -5292.795} C_VEL
LIN {X 0,Y 427.939,Z 837.306,A -85,B 0,C 180,E1 -5294.969,E2 -5294.969} C_VEL
LIN {X 0,Y 426.854,Z 846.527,A -85,B 0,C 180,E1 -5297.28,E2 -5297.28} C_VEL
LIN {X 0,Y 426.001,Z 854.218,A -85,B 0,C 180,E1 -5299.725,E2 -5299.725} C_VEL
LIN {X 0,Y 425.448,Z 860.038,A -85,B 0,C 180,E1 -5302.166,E2 -5302.166} C_VEL
LIN {X 0,Y 425.128,Z 864.167,A -85,B 0,C 180,E1 -5304.602,E2 -5304.602} C_VEL
LIN {X 0,Y 424.945,Z 866.841,A -85,B 0,C 180,E1 -5307.168,E2 -5307.168} C_VEL
LIN {X 0,Y 424.885,Z 867.86,A -85,B 0,C 180,E1 -5309.731,E2 -5309.731} C_VEL
LIN {X 0,Y 424.923,Z 867.253,A -85,B 0,C 180,E1 -5312.293,E2 -5312.293} C_VEL
LIN {X 0,Y 425.083,Z 865.004,A -85,B 0,C 180,E1 -5314.858,E2 -5314.858} C_VEL
LIN {X 0,Y 425.379,Z 861.049,A -85,B 0,C 180,E1 -5317.428,E2 -5317.428} C_VEL
LIN {X 0,Y 425.908,Z 855.226,A -85,B 0,C 180,E1 -5320.005,E2 -5320.005} C_VEL
LIN {X 0,Y 426.711,Z 847.816,A -85,B 0,C 180,E1 -5322.45,E2 -5322.45} C_VEL
LIN {X 0,Y 427.751,Z 838.9,A -85,B 0,C 180,E1 -5324.761,E2 -5324.761} C_VEL
LIN {X 0,Y 429.039,Z 828.498,A -85,B 0,C 180,E1 -5326.937,E2 -5326.937} C_VEL
LIN {X 0,Y 430.546,Z 816.592,A -85,B 0,C 180,E1 -5328.973,E2 -5328.973} C_VEL
LIN {X 0,Y 432.194,Z 803.092,A -85,B 0,C 180,E1 -5330.872,E2 -5330.872} C_VEL
LIN {X 0,Y 433.88,Z 788.439,A -85,B 0,C 180,E1 -5332.563,E2 -5332.563} C_VEL
LIN {X 0,Y 435.403,Z 773.445,A -85,B 0,C 180,E1 -5333.983,E2 -5333.983} C_VEL
LIN {X 0,Y 436.803,Z 757.671,A -85,B 0,C 180,E1 -5335.199,E2 -5335.199} C_VEL
LIN {X 0,Y 438.015,Z 741.071,A -85,B 0,C 180,E1 -5336.219,E2 -5336.219} C_VEL
LIN {X 0,Y 438.97,Z 723.208,A -85,B 0,C 180,E1 -5337.06,E2 -5337.06} C_VEL
LIN {X 0,Y 439.562,Z 704.747,A -85,B 0,C 180,E1 -5337.68,E2 -5337.68} C_VEL
LIN {X 0,Y 439.88,Z 682.054,A -85,B 0,C 180,E1 -5338.147,E2 -5338.147} C_VEL
LIN {X 0,Y 443.467,Z 497.403,A -85,B 0,C 180,E1 -5341.302,E2 -5341.302} C_VEL
LIN {X 0,Y 442.527,Z 490.584,A -85,B 0,C 180,E1 -5341.538,E2 -5341.538} C_VEL
LIN {X 0,Y 443.479,Z 457.94,A -85,B 0,C 180,E1 -5343.933,E2 -5343.933} C_VEL
LIN {X 0,Y 445.043,Z 425.333,A -85,B 0,C 180,E1 -5346.513,E2 -5346.513} C_VEL
LIN {X 0,Y 437.79,Z 406.01,A -85,B 0,C 180,E1 -5348.908,E2 -5348.908} C_VEL
LIN {X 0,Y 430.079,Z 388.508,A -85,B 0,C 180,E1 -5351.229,E2 -5351.229} C_VEL
LIN {X 0,Y 426.633,Z 381.332,A -85,B 0,C 180,E1 -5352.219,E2 -5352.219} C_VEL
LIN {X 0,Y 425.278,Z 377.774,A -85,B 0,C 180,E1 -5352.669,E2 -5352.669} C_VEL
LIN {X 0,Y 425.323,Z 377.889,A -85,B 0,C 180,E1 -5353.063,E2 -5353.063} C_VEL
LIN {X 0,Y 426.854,Z 381.591,A -85,B 0,C 180,E1 -5353.71,E2 -5353.71} C_VEL
LIN {X 0,Y 434.295,Z 397.702,A -85,B 0,C 180,E1 -5356.498,E2 -5356.498} C_VEL
LIN {X 0,Y 442.555,Z 417.263,A -85,B 0,C 180,E1 -5359.587,E2 -5359.587} C_VEL
LIN {X 0,Y 448.088,Z 432.134,A -85,B 0,C 180,E1 -5361.741,E2 -5361.741} C_VEL
LIN {X 0,Y 444.578,Z 473.076,A -85,B 0,C 180,E1 -5365.476,E2 -5365.476} C_VEL
LIN {X 0,Y 441.146,Z 515.955,A -85,B 0,C 180,E1 -5369.338,E2 -5369.338} C_VEL
LIN {X 0,Y 437.96,Z 560.346,A -85,B 0,C 180,E1 -5373.272,E2 -5373.272} C_VEL
LIN {X 0,Y 435.461,Z 601.367,A -85,B 0,C 180,E1 -5376.825,E2 -5376.825} C_VEL
LIN {X 0,Y 436.225,Z 609.77,A -85,B 0,C 180,E1 -5377.071,E2 -5377.071} C_VEL
LIN {X 0,Y 432.199,Z 747.454,A -85,B 0,C 180,E1 -5380.057,E2 -5380.057} C_VEL
LIN {X 0,Y 431.728,Z 764.757,A -85,B 0,C 180,E1 -5380.693,E2 -5380.693} C_VEL
LIN {X 0,Y 431.101,Z 779.624,A -85,B 0,C 180,E1 -5381.473,E2 -5381.473} C_VEL
LIN {X 0,Y 430.259,Z 795.147,A -85,B 0,C 180,E1 -5382.555,E2 -5382.555} C_VEL
LIN {X 0,Y 429.378,Z 808.858,A -85,B 0,C 180,E1 -5383.773,E2 -5383.773} C_VEL
LIN {X 0,Y 428.392,Z 822.733,A -85,B 0,C 180,E1 -5385.33,E2 -5385.33} C_VEL
LIN {X 0,Y 427.563,Z 833.919,A -85,B 0,C 180,E1 -5386.889,E2 -5386.889} C_VEL
LIN {X 0,Y 426.759,Z 844.819,A -85,B 0,C 180,E1 -5388.786,E2 -5388.786} C_VEL
LIN {X 0,Y 426.163,Z 853.461,A -85,B 0,C 180,E1 -5390.683,E2 -5390.683} C_VEL
LIN {X 0,Y 425.703,Z 861.05,A -85,B 0,C 180,E1 -5392.849,E2 -5392.849} C_VEL
LIN {X 0,Y 425.439,Z 866.274,A -85,B 0,C 180,E1 -5394.876,E2 -5394.876} C_VEL
LIN {X 0,Y 425.326,Z 870.221,A -85,B 0,C 180,E1 -5397.17,E2 -5397.17} C_VEL
LIN {X 0,Y 425.324,Z 872.166,A -85,B 0,C 180,E1 -5399.326,E2 -5399.326} C_VEL
LIN {X 0,Y 425.455,Z 872.401,A -85,B 0,C 180,E1 -5401.616,E2 -5401.616} C_VEL
LIN {X 0,Y 425.674,Z 870.897,A -85,B 0,C 180,E1 -5403.771,E2 -5403.771} C_VEL
LIN {X 0,Y 426.098,Z 867.442,A -85,B 0,C 180,E1 -5406.061,E2 -5406.061} C_VEL
LIN {X 0,Y 426.637,Z 862.622,A -85,B 0,C 180,E1 -5408.083,E2 -5408.083} C_VEL
LIN {X 0,Y 427.405,Z 856.026,A -85,B 0,C 180,E1 -5410.105,E2 -5410.105} C_VEL
LIN {X 0,Y 428.302,Z 847.933,A -85,B 0,C 180,E1 -5411.999,E2 -5411.999} C_VEL
LIN {X 0,Y 429.423,Z 837.721,A -85,B 0,C 180,E1 -5413.876,E2 -5413.876} C_VEL
LIN {X 0,Y 430.612,Z 826.024,A -85,B 0,C 180,E1 -5415.556,E2 -5415.556} C_VEL
LIN {X 0,Y 431.754,Z 813.733,A -85,B 0,C 180,E1 -5416.974,E2 -5416.974} C_VEL
LIN {X 0,Y 432.837,Z 799.861,A -85,B 0,C 180,E1 -5418.24,E2 -5418.24} C_VEL
LIN {X 0,Y 433.698,Z 785.65,A -85,B 0,C 180,E1 -5419.249,E2 -5419.249} C_VEL
LIN {X 0,Y 434.381,Z 770.694,A -85,B 0,C 180,E1 -5420.057,E2 -5420.057} C_VEL
LIN {X 0,Y 434.933,Z 750.648,A -85,B 0,C 180,E1 -5420.804,E2 -5420.804} C_VEL
LIN {X 0,Y 438.029,Z 707.841,A -85,B 0,C 180,E1 -5422.215,E2 -5422.215} C_VEL
LIN {X 0,Y 446.109,Z 628.568,A -85,B 0,C 180,E1 -5424.818,E2 -5424.818} C_VEL
LIN {X 0,Y 450.298,Z 617.441,A -85,B 0,C 180,E1 -5425.586,E2 -5425.586} C_VEL
LIN {X 0,Y 457.37,Z 584.403,A -85,B 0,C 180,E1 -5429.104,E2 -5429.104} C_VEL
LIN {X 0,Y 465.099,Z 558.297,A -85,B 0,C 180,E1 -5432.072,E2 -5432.072} C_VEL
LIN {X 0,Y 472.793,Z 539.414,A -85,B 0,C 180,E1 -5434.378,E2 -5434.378} C_VEL
LIN {X 0,Y 479.156,Z 527.582,A -85,B 0,C 180,E1 -5435.938,E2 -5435.938} C_VEL
LIN {X 0,Y 474.72,Z 536.179,A -85,B 0,C 180,E1 -5437.435,E2 -5437.435} C_VEL
LIN {X 0,Y 472.589,Z 544.537,A -85,B 0,C 180,E1 -5438.929,E2 -5438.929} C_VEL
LIN {X 0,Y 472.602,Z 552.68,A -85,B 0,C 180,E1 -5440.391,E2 -5440.391} C_VEL
LIN {X 0,Y 474.713,Z 561.114,A -85,B 0,C 180,E1 -5441.888,E2 -5441.888} C_VEL
LIN {X 0,Y 479.191,Z 570.046,A -85,B 0,C 180,E1 -5443.437,E2 -5443.437} C_VEL
LIN {X 0,Y 486.332,Z 579.294,A -85,B 0,C 180,E1 -5445.01,E2 -5445.01} C_VEL
LIN {X 0,Y 495.376,Z 587.742,A -85,B 0,C 180,E1 -5446.435,E2 -5446.435} C_VEL
LIN {X 0,Y 501.797,Z 592.738,A -85,B 0,C 180,E1 -5447.25,E2 -5447.25} C_VEL
LIN {X 0,Y 486.17,Z 619.263,A -85,B 0,C 180,E1 -5447.818,E2 -5447.818} C_VEL
LIN {X 0,Y 475.81,Z 639.636,A -85,B 0,C 180,E1 -5448.391,E2 -5448.391} C_VEL
LIN {X 0,Y 468.721,Z 656.707,A -85,B 0,C 180,E1 -5449.008,E2 -5449.008} C_VEL
LIN {X 0,Y 459.615,Z 677.671,A -85,B 0,C 180,E1 -5449.751,E2 -5449.751} C_VEL
LIN {X 0,Y 450.187,Z 705.587,A -85,B 0,C 180,E1 -5450.975,E2 -5450.975} C_VEL
LIN {X 0,Y 449.607,Z 708.714,A -85,B 0,C 180,E1 -5451.069,E2 -5451.069} C_VEL
LIN {X 0,Y 448.076,Z 724.952,A -85,B 0,C 180,E1 -5451.301,E2 -5451.301} C_VEL
LIN {X 0,Y 446.954,Z 755.184,A -85,B 0,C 180,E1 -5451.935,E2 -5451.935} C_VEL
LIN {X 0,Y 445.305,Z 779.469,A -85,B 0,C 180,E1 -5452.67,E2 -5452.67} C_VEL
LIN {X 0,Y 443.467,Z 803.048,A -85,B 0,C 180,E1 -5453.631,E2 -5453.631} C_VEL
LIN {X 0,Y 441.455,Z 825.873,A -85,B 0,C 180,E1 -5454.808,E2 -5454.808} C_VEL
LIN {X 0,Y 439.319,Z 847.555,A -85,B 0,C 180,E1 -5456.188,E2 -5456.188} C_VEL
LIN {X 0,Y 437.077,Z 869.358,A -85,B 0,C 180,E1 -5457.859,E2 -5457.859} C_VEL
LIN {X 0,Y 434.938,Z 888.742,A -85,B 0,C 180,E1 -5459.619,E2 -5459.619} C_VEL
LIN {X 0,Y 432.86,Z 907.149,A -85,B 0,C 180,E1 -5461.586,E2 -5461.586} C_VEL
LIN {X 0,Y 430.998,Z 923.321,A -85,B 0,C 180,E1 -5463.607,E2 -5463.607} C_VEL
LIN {X 0,Y 429.186,Z 939.276,A -85,B 0,C 180,E1 -5465.94,E2 -5465.94} C_VEL
LIN {X 0,Y 427.587,Z 953.85,A -85,B 0,C 180,E1 -5468.461,E2 -5468.461} C_VEL
LIN {X 0,Y 426.285,Z 966.662,A -85,B 0,C 180,E1 -5471.114,E2 -5471.114} C_VEL
LIN {X 0,Y 425.393,Z 976.757,A -85,B 0,C 180,E1 -5473.617,E2 -5473.617} C_VEL
LIN {X 0,Y 424.686,Z 985.971,A -85,B 0,C 180,E1 -5476.382,E2 -5476.382} C_VEL
LIN {X 0,Y 424.249,Z 993.558,A -85,B 0,C 180,E1 -5479.269,E2 -5479.269} C_VEL
LIN {X 0,Y 424.001,Z 999.166,A -85,B 0,C 180,E1 -5482.138,E2 -5482.138} C_VEL
LIN {X 0,Y 423.915,Z 1002.704,A -85,B 0,C 180,E1 -5484.722,E2 -5484.722} C_VEL
LIN {X 0,Y 423.901,Z 1004.859,A -85,B 0,C 180,E1 -5487.566,E2 -5487.566} C_VEL
LIN {X 0,Y 423.894,Z 1005.408,A -85,B 0,C 180,E1 -5490.675,E2 -5490.675} C_VEL
LIN {X 0,Y 423.909,Z 1004.348,A -85,B 0,C 180,E1 -5493.38,E2 -5493.38} C_VEL
LIN {X 0,Y 423.953,Z 1001.574,A -85,B 0,C 180,E1 -5496.228,E2 -5496.228} C_VEL
LIN {X 0,Y 424.084,Z 997.035,A -85,B 0,C 180,E1 -5499.088,E2 -5499.088} C_VEL
LIN {X 0,Y 424.37,Z 991.076,A -85,B 0,C 180,E1 -5501.828,E2 -5501.828} C_VEL
LIN {X 0,Y 424.895,Z 982.91,A -85,B 0,C 180,E1 -5504.726,E2 -5504.726} C_VEL
LIN {X 0,Y 425.739,Z 973.036,A -85,B 0,C 180,E1 -5507.542,E2 -5507.542} C_VEL
LIN {X 0,Y 426.921,Z 961.421,A -85,B 0,C 180,E1 -5510.28,E2 -5510.28} C_VEL
LIN {X 0,Y 428.363,Z 948.761,A -85,B 0,C 180,E1 -5512.797,E2 -5512.797} C_VEL
LIN {X 0,Y 430.22,Z 933.852,A -85,B 0,C 180,E1 -5515.317,E2 -5515.317} C_VEL
LIN {X 0,Y 432.415,Z 917.293,A -85,B 0,C 180,E1 -5517.695,E2 -5517.695} C_VEL
LIN {X 0,Y 434.884,Z 898.974,A -85,B 0,C 180,E1 -5519.928,E2 -5519.928} C_VEL
LIN {X 0,Y 437.575,Z 878.612,A -85,B 0,C 180,E1 -5522.013,E2 -5522.013} C_VEL
LIN {X 0,Y 440.045,Z 859.518,A -85,B 0,C 180,E1 -5523.67,E2 -5523.67} C_VEL
LIN {X 0,Y 442.455,Z 839.589,A -85,B 0,C 180,E1 -5525.111,E2 -5525.111} C_VEL
LIN {X 0,Y 444.864,Z 818.149,A -85,B 0,C 180,E1 -5526.395,E2 -5526.395} C_VEL
LIN {X 0,Y 446.887,Z 797.698,A -85,B 0,C 180,E1 -5527.383,E2 -5527.383} C_VEL
LIN {X 0,Y 448.715,Z 775.665,A -85,B 0,C 180,E1 -5528.2,E2 -5528.2} C_VEL
LIN {X 0,Y 450.23,Z 752.822,A -85,B 0,C 180,E1 -5528.812,E2 -5528.812} C_VEL
LIN {X 0,Y 451.676,Z 717.254,A -85,B 0,C 180,E1 -5529.469,E2 -5529.469} C_VEL
LIN {X 0,Y 452.223,Z 713.393,A -85,B 0,C 180,E1 -5529.551,E2 -5529.551} C_VEL
LIN {X 0,Y 457.494,Z 697.094,A -85,B 0,C 180,E1 -5530.309,E2 -5530.309} C_VEL
LIN {X 0,Y 464.882,Z 676.96,A -85,B 0,C 180,E1 -5531.158,E2 -5531.158} C_VEL
LIN {X 0,Y 472.828,Z 659.107,A -85,B 0,C 180,E1 -5531.767,E2 -5531.767} C_VEL
LIN {X 0,Y 480.131,Z 641.998,A -85,B 0,C 180,E1 -5532.365,E2 -5532.365} C_VEL
LIN {X 0,Y 490.555,Z 621.657,A -85,B 0,C 180,E1 -5532.903,E2 -5532.903} C_VEL
LIN {X 0,Y 505.54,Z 595.738,A -85,B 0,C 180,E1 -5533.413,E2 -5533.413} C_VEL
LIN {X 0,Y 494.912,Z 587.098,A -85,B 0,C 180,E1 -5535.001,E2 -5535.001} C_VEL
LIN {X 0,Y 485.62,Z 576.489,A -85,B 0,C 180,E1 -5536.716,E2 -5536.716} C_VEL
LIN {X 0,Y 478.922,Z 565.912,A -85,B 0,C 180,E1 -5538.243,E2 -5538.243} C_VEL
LIN {X 0,Y 473.138,Z 552.783,A -85,B 0,C 180,E1 -5539.948,E2 -5539.948} C_VEL
LIN {X 0,Y 469.198,Z 538.567,A -85,B 0,C 180,E1 -5541.598,E2 -5541.598} C_VEL
LIN {X 0,Y 466.951,Z 523.074,A -85,B 0,C 180,E1 -5543.209,E2 -5543.209} C_VEL
LIN {X 0,Y 466.36,Z 504.699,A -85,B 0,C 180,E1 -5544.93,E2 -5544.93} C_VEL
LIN {X 0,Y 467.769,Z 483.323,A -85,B 0,C 180,E1 -5546.695,E2 -5546.695} C_VEL
LIN {X 0,Y 470.643,Z 458.568,A -85,B 0,C 180,E1 -5548.635,E2 -5548.635} C_VEL
LIN {X 0,Y 460.888,Z 440.473,A -85,B 0,C 180,E1 -5551.917,E2 -5551.917} C_VEL
LIN {X 0,Y 453.215,Z 426.66,A -85,B 0,C 180,E1 -5554.66,E2 -5554.66} C_VEL
LIN {X 0,Y 445.234,Z 412.536,A -85,B 0,C 180,E1 -5557.696,E2 -5557.696} C_VEL
LIN {X 0,Y 439.322,Z 402.487,A -85,B 0,C 180,E1 -5560.039,E2 -5560.039} C_VEL
LIN {X 0,Y 436.614,Z 397.783,A -85,B 0,C 180,E1 -5561.162,E2 -5561.162} C_VEL
LIN {X 0,Y 433.684,Z 392.718,A -85,B 0,C 180,E1 -5562.421,E2 -5562.421} C_VEL
LIN {X 0,Y 431.422,Z 388.635,A -85,B 0,C 180,E1 -5563.438,E2 -5563.438} C_VEL
LIN {X 0,Y 428.765,Z 384.472,A -85,B 0,C 180,E1 -5564.583,E2 -5564.583} C_VEL
LIN {X 0,Y 428.019,Z 382.807,A -85,B 0,C 180,E1 -5564.972,E2 -5564.972} C_VEL
LIN {X 0,Y 425.86,Z 379.873,A -85,B 0,C 180,E1 -5565.867,E2 -5565.867} C_VEL
LIN {X 0,Y 425.306,Z 377.753,A -85,B 0,C 180,E1 -5566.331,E2 -5566.331} C_VEL
LIN {X 0,Y 425.318,Z 377.753,A -85,B 0,C 180,E1 -5570.256,E2 -5570.256} C_VEL
LIN {X 0,Y 425.282,Z 377.758,A -85,B 0,C 180,E1 -5574.063,E2 -5574.063} C_VEL
LIN {X 0,Y 425.306,Z 377.76,A -85,B 0,C 180,E1 -5577.98,E2 -5577.98} C_VEL
LIN {X 0,Y 425.299,Z 377.765,A -85,B 0,C 180,E1 -5581.617,E2 -5581.617} C_VEL
LIN {X 0,Y 425.306,Z 377.757,A -85,B 0,C 180,E1 -5585.532,E2 -5585.532} C_VEL
LIN {X 0,Y 425.309,Z 377.762,A -85,B 0,C 180,E1 -5589.199,E2 -5589.199} C_VEL
LIN {X 0,Y 425.32,Z 377.754,A -85,B 0,C 180,E1 -5593.043,E2 -5593.043} C_VEL
LIN {X 0,Y 425.28,Z 377.761,A -85,B 0,C 180,E1 -5596.887,E2 -5596.887} C_VEL
LIN {X 0,Y 425.313,Z 377.753,A -85,B 0,C 180,E1 -5600.793,E2 -5600.793} C_VEL
LIN {X 0,Y 425.288,Z 377.759,A -85,B 0,C 180,E1 -5604.517,E2 -5604.517} C_VEL
LIN {X 0,Y 425.307,Z 377.753,A -85,B 0,C 180,E1 -5608.505,E2 -5608.505} C_VEL
LIN {X 0,Y 425.31,Z 377.752,A -85,B 0,C 180,E1 -5612.253,E2 -5612.253} C_VEL
LIN {X 0,Y 425.316,Z 377.716,A -85,B 0,C 180,E1 -5616.162,E2 -5616.162} C_VEL
LIN {X 0,Y 425.285,Z 377.762,A -85,B 0,C 180,E1 -5619.929,E2 -5619.929} C_VEL
LIN {X 0,Y 425.315,Z 377.739,A -85,B 0,C 180,E1 -5623.722,E2 -5623.722} C_VEL
LIN {X 0,Y 425.301,Z 377.931,A -85,B 0,C 180,E1 -5627.452,E2 -5627.452} C_VEL
LIN {X 0,Y 426.377,Z 380.911,A -85,B 0,C 180,E1 -5627.819,E2 -5627.819} C_VEL
LIN {X 0,Y 427.883,Z 383.913,A -85,B 0,C 180,E1 -5628.243,E2 -5628.243} C_VEL
LIN {X 0,Y 435.271,Z 399.917,A -85,B 0,C 180,E1 -5630.415,E2 -5630.415} C_VEL
LIN {X 0,Y 442.824,Z 419.245,A -85,B 0,C 180,E1 -5632.849,E2 -5632.849} C_VEL
LIN {X 0,Y 445.054,Z 425.765,A -85,B 0,C 180,E1 -5633.623,E2 -5633.623} C_VEL
LIN {X 0,Y 443.104,Z 467.72,A -85,B 0,C 180,E1 -5636.903,E2 -5636.903} C_VEL
LIN {X 0,Y 442.564,Z 491.594,A -85,B 0,C 180,E1 -5638.611,E2 -5638.611} C_VEL
LIN {X 0,Y 443.583,Z 499.943,A -85,B 0,C 180,E1 -5638.851,E2 -5638.851} C_VEL
LIN {X 0,Y 440.496,Z 649.066,A -85,B 0,C 180,E1 -5641.386,E2 -5641.386} C_VEL
LIN {X 0,Y 439.498,Z 656.749,A -85,B 0,C 180,E1 -5641.454,E2 -5641.454} C_VEL
LIN {X 0,Y 433.639,Z 677.174,A -85,B 0,C 180,E1 -5641.397,E2 -5641.397} C_VEL
LIN {X 0,Y 432.861,Z 683.769,A -85,B 0,C 180,E1 -5641.462,E2 -5641.462} C_VEL
LIN {X 0,Y 432.531,Z 706.042,A -85,B 0,C 180,E1 -5641.929,E2 -5641.929} C_VEL
LIN {X 0,Y 431.915,Z 724.514,A -85,B 0,C 180,E1 -5642.56,E2 -5642.56} C_VEL
LIN {X 0,Y 430.938,Z 742.059,A -85,B 0,C 180,E1 -5643.398,E2 -5643.398} C_VEL
LIN {X 0,Y 429.583,Z 759.587,A -85,B 0,C 180,E1 -5644.495,E2 -5644.495} C_VEL
LIN {X 0,Y 428.047,Z 776.008,A -85,B 0,C 180,E1 -5645.799,E2 -5645.799} C_VEL
LIN {X 0,Y 426.372,Z 791.406,A -85,B 0,C 180,E1 -5647.31,E2 -5647.31} C_VEL
LIN {X 0,Y 424.619,Z 805.765,A -85,B 0,C 180,E1 -5649.028,E2 -5649.028} C_VEL
LIN {X 0,Y 422.904,Z 819.027,A -85,B 0,C 180,E1 -5650.958,E2 -5650.958} C_VEL
LIN {X 0,Y 421.333,Z 830.734,A -85,B 0,C 180,E1 -5653.029,E2 -5653.029} C_VEL
LIN {X 0,Y 419.988,Z 840.962,A -85,B 0,C 180,E1 -5655.243,E2 -5655.243} C_VEL
LIN {X 0,Y 418.901,Z 849.722,A -85,B 0,C 180,E1 -5657.596,E2 -5657.596} C_VEL
LIN {X 0,Y 418.057,Z 856.971,A -85,B 0,C 180,E1 -5660.085,E2 -5660.085} C_VEL
LIN {X 0,Y 417.495,Z 862.628,A -85,B 0,C 180,E1 -5662.708,E2 -5662.708} C_VEL
LIN {X 0,Y 417.183,Z 866.461,A -85,B 0,C 180,E1 -5665.326,E2 -5665.326} C_VEL
LIN {X 0,Y 417.019,Z 868.597,A -85,B 0,C 180,E1 -5667.939,E2 -5667.939} C_VEL
LIN {X 0,Y 416.983,Z 869.095,A -85,B 0,C 180,E1 -5670.55,E2 -5670.55} C_VEL
LIN {X 0,Y 417.069,Z 867.862,A -85,B 0,C 180,E1 -5673.299,E2 -5673.299} C_VEL
LIN {X 0,Y 417.289,Z 864.988,A -85,B 0,C 180,E1 -5675.914,E2 -5675.914} C_VEL
LIN {X 0,Y 417.672,Z 860.645,A -85,B 0,C 180,E1 -5678.397,E2 -5678.397} C_VEL
LIN {X 0,Y 418.312,Z 854.601,A -85,B 0,C 180,E1 -5680.885,E2 -5680.885} C_VEL
LIN {X 0,Y 419.258,Z 846.791,A -85,B 0,C 180,E1 -5683.34,E2 -5683.34} C_VEL
LIN {X 0,Y 420.491,Z 837.173,A -85,B 0,C 180,E1 -5685.729,E2 -5685.729} C_VEL
LIN {X 0,Y 421.977,Z 826.091,A -85,B 0,C 180,E1 -5687.941,E2 -5687.941} C_VEL
LIN {X 0,Y 423.545,Z 814.308,A -85,B 0,C 180,E1 -5689.874,E2 -5689.874} C_VEL
LIN {X 0,Y 425.292,Z 800.552,A -85,B 0,C 180,E1 -5691.733,E2 -5691.733} C_VEL
LIN {X 0,Y 426.974,Z 786.397,A -85,B 0,C 180,E1 -5693.313,E2 -5693.313} C_VEL
LIN {X 0,Y 428.595,Z 770.639,A -85,B 0,C 180,E1 -5694.756,E2 -5694.756} C_VEL
LIN {X 0,Y 430.049,Z 754.247,A -85,B 0,C 180,E1 -5695.965,E2 -5695.965} C_VEL
LIN {X 0,Y 431.26,Z 737.197,A -85,B 0,C 180,E1 -5696.953,E2 -5696.953} C_VEL
LIN {X 0,Y 432.146,Z 719.01,A -85,B 0,C 180,E1 -5697.747,E2 -5697.747} C_VEL
LIN {X 0,Y 432.667,Z 700.041,A -85,B 0,C 180,E1 -5698.314,E2 -5698.314} C_VEL
LIN {X 0,Y 434.723,Z 595.727,A -85,B 0,C 180,E1 -5700.149,E2 -5700.149} C_VEL
LIN {X 0,Y 436.676,Z 498.539,A -85,B 0,C 180,E1 -5701.844,E2 -5701.844} C_VEL
LIN {X 0,Y 435.765,Z 491.756,A -85,B 0,C 180,E1 -5702.085,E2 -5702.085} C_VEL
LIN {X 0,Y 436.779,Z 458.993,A -85,B 0,C 180,E1 -5704.502,E2 -5704.502} C_VEL
LIN {X 0,Y 438.288,Z 428.66,A -85,B 0,C 180,E1 -5706.908,E2 -5706.908} C_VEL
LIN {X 0,Y 431.291,Z 409.961,A -85,B 0,C 180,E1 -5709.265,E2 -5709.265} C_VEL
LIN {X 0,Y 424.109,Z 393.465,A -85,B 0,C 180,E1 -5711.489,E2 -5711.489} C_VEL
LIN {X 0,Y 419.436,Z 383.523,A -85,B 0,C 180,E1 -5712.901,E2 -5712.901} C_VEL
LIN {X 0,Y 426.857,Z 399.761,A -85,B 0,C 180,E1 -5715.789,E2 -5715.789} C_VEL
LIN {X 0,Y 434.124,Z 416.767,A -85,B 0,C 180,E1 -5718.563,E2 -5718.563} C_VEL
LIN {X 0,Y 441.318,Z 435.319,A -85,B 0,C 180,E1 -5721.34,E2 -5721.34} C_VEL
LIN {X 0,Y 437.628,Z 476.171,A -85,B 0,C 180,E1 -5725.107,E2 -5725.107} C_VEL
LIN {X 0,Y 434.047,Z 519.148,A -85,B 0,C 180,E1 -5729.012,E2 -5729.012} C_VEL
LIN {X 0,Y 430.681,Z 563.806,A -85,B 0,C 180,E1 -5733.015,E2 -5733.015} C_VEL
LIN {X 0,Y 428.214,Z 602.119,A -85,B 0,C 180,E1 -5736.37,E2 -5736.37} C_VEL
LIN {X 0,Y 428.989,Z 610.801,A -85,B 0,C 180,E1 -5736.63,E2 -5736.63} C_VEL
LIN {X 0,Y 424.671,Z 748.395,A -85,B 0,C 180,E1 -5739.71,E2 -5739.71} C_VEL
LIN {X 0,Y 424.195,Z 765.058,A -85,B 0,C 180,E1 -5740.332,E2 -5740.332} C_VEL
LIN {X 0,Y 423.479,Z 781.277,A -85,B 0,C 180,E1 -5741.199,E2 -5741.199} C_VEL
LIN {X 0,Y 422.605,Z 796.667,A -85,B 0,C 180,E1 -5742.3,E2 -5742.3} C_VEL
LIN {X 0,Y 421.691,Z 810.175,A -85,B 0,C 180,E1 -5743.528,E2 -5743.528} C_VEL
LIN {X 0,Y 420.653,Z 824.125,A -85,B 0,C 180,E1 -5745.125,E2 -5745.125} C_VEL
LIN {X 0,Y 419.749,Z 835.701,A -85,B 0,C 180,E1 -5746.78,E2 -5746.78} C_VEL
LIN {X 0,Y 418.918,Z 846.536,A -85,B 0,C 180,E1 -5748.713,E2 -5748.713} C_VEL
LIN {X 0,Y 418.296,Z 855.079,A -85,B 0,C 180,E1 -5750.645,E2 -5750.645} C_VEL
LIN {X 0,Y 417.822,Z 862.635,A -85,B 0,C 180,E1 -5752.851,E2 -5752.851} C_VEL
LIN {X 0,Y 417.536,Z 868.067,A -85,B 0,C 180,E1 -5755.054,E2 -5755.054} C_VEL
LIN {X 0,Y 417.44,Z 871.711,A -85,B 0,C 180,E1 -5757.254,E2 -5757.254} C_VEL
LIN {X 0,Y 417.447,Z 873.596,A -85,B 0,C 180,E1 -5759.451,E2 -5759.451} C_VEL
LIN {X 0,Y 417.602,Z 873.815,A -85,B 0,C 180,E1 -5761.783,E2 -5761.783} C_VEL
LIN {X 0,Y 417.853,Z 872.244,A -85,B 0,C 180,E1 -5763.979,E2 -5763.979} C_VEL
LIN {X 0,Y 418.297,Z 869.011,A -85,B 0,C 180,E1 -5766.175,E2 -5766.175} C_VEL
LIN {X 0,Y 418.932,Z 863.891,A -85,B 0,C 180,E1 -5768.371,E2 -5768.371} C_VEL
LIN {X 0,Y 419.789,Z 857.287,A -85,B 0,C 180,E1 -5770.429,E2 -5770.429} C_VEL
LIN {X 0,Y 420.802,Z 848.783,A -85,B 0,C 180,E1 -5772.426,E2 -5772.426} C_VEL
LIN {X 0,Y 421.983,Z 838.837,A -85,B 0,C 180,E1 -5774.265,E2 -5774.265} C_VEL
LIN {X 0,Y 423.285,Z 827.172,A -85,B 0,C 180,E1 -5775.971,E2 -5775.971} C_VEL
LIN {X 0,Y 424.491,Z 814.834,A -85,B 0,C 180,E1 -5777.406,E2 -5777.406} C_VEL
LIN {X 0,Y 425.68,Z 800.916,A -85,B 0,C 180,E1 -5778.7,E2 -5778.7} C_VEL
LIN {X 0,Y 426.669,Z 785.568,A -85,B 0,C 180,E1 -5779.793,E2 -5779.793} C_VEL
LIN {X 0,Y 427.391,Z 769.941,A -85,B 0,C 180,E1 -5780.622,E2 -5780.622} C_VEL
LIN {X 0,Y 428.689,Z 740.393,A -85,B 0,C 180,E1 -5781.722,E2 -5781.722} C_VEL
LIN {X 0,Y 439.403,Z 638.018,A -85,B 0,C 180,E1 -5785.255,E2 -5785.255} C_VEL
LIN {X 0,Y 440.305,Z 631.312,A -85,B 0,C 180,E1 -5785.488,E2 -5785.488} C_VEL
LIN {X 0,Y 444.834,Z 619.73,A -85,B 0,C 180,E1 -5786.282,E2 -5786.282} C_VEL
LIN {X 0,Y 452.204,Z 588.529,A -85,B 0,C 180,E1 -5789.688,E2 -5789.688} C_VEL
LIN {X 0,Y 460.072,Z 564.23,A -85,B 0,C 180,E1 -5792.517,E2 -5792.517} C_VEL
LIN {X 0,Y 468.083,Z 546.149,A -85,B 0,C 180,E1 -5794.773,E2 -5794.773} C_VEL
LIN {X 0,Y 473.431,Z 536.749,A -85,B 0,C 180,E1 -5796.013,E2 -5796.013} C_VEL
LIN {X 0,Y 469.426,Z 544.957,A -85,B 0,C 180,E1 -5797.529,E2 -5797.529} C_VEL
LIN {X 0,Y 467.669,Z 552.89,A -85,B 0,C 180,E1 -5799.022,E2 -5799.022} C_VEL
LIN {X 0,Y 468.032,Z 561.175,A -85,B 0,C 180,E1 -5800.579,E2 -5800.579} C_VEL
LIN {X 0,Y 470.664,Z 569.782,A -85,B 0,C 180,E1 -5802.167,E2 -5802.167} C_VEL
LIN {X 0,Y 475.669,Z 578.566,A -85,B 0,C 180,E1 -5803.753,E2 -5803.753} C_VEL
LIN {X 0,Y 483.387,Z 587.736,A -85,B 0,C 180,E1 -5805.36,E2 -5805.36} C_VEL
LIN {X 0,Y 492.65,Z 595.99,A -85,B 0,C 180,E1 -5806.769,E2 -5806.769} C_VEL
LIN {X 0,Y 478.446,Z 620.697,A -85,B 0,C 180,E1 -5807.301,E2 -5807.301} C_VEL
LIN {X 0,Y 468.707,Z 640.276,A -85,B 0,C 180,E1 -5807.863,E2 -5807.863} C_VEL
LIN {X 0,Y 460.712,Z 659.336,A -85,B 0,C 180,E1 -5808.553,E2 -5808.553} C_VEL
LIN {X 0,Y 452.908,Z 677.37,A -85,B 0,C 180,E1 -5809.196,E2 -5809.196} C_VEL
LIN {X 0,Y 443.363,Z 705.628,A -85,B 0,C 180,E1 -5810.438,E2 -5810.438} C_VEL
LIN {X 0,Y 441.448,Z 724.981,A -85,B 0,C 180,E1 -5810.721,E2 -5810.721} C_VEL
LIN {X 0,Y 440.171,Z 754.528,A -85,B 0,C 180,E1 -5811.376,E2 -5811.376} C_VEL
LIN {X 0,Y 438.257,Z 779.928,A -85,B 0,C 180,E1 -5812.183,E2 -5812.183} C_VEL
LIN {X 0,Y 436.2,Z 804.123,A -85,B 0,C 180,E1 -5813.213,E2 -5813.213} C_VEL
LIN {X 0,Y 434.028,Z 826.604,A -85,B 0,C 180,E1 -5814.431,E2 -5814.431} C_VEL
LIN {X 0,Y 431.572,Z 849.904,A -85,B 0,C 180,E1 -5815.978,E2 -5815.978} C_VEL
LIN {X 0,Y 429.253,Z 871.232,A -85,B 0,C 180,E1 -5817.684,E2 -5817.684} C_VEL
LIN {X 0,Y 426.894,Z 891.378,A -85,B 0,C 180,E1 -5819.608,E2 -5819.608} C_VEL
LIN {X 0,Y 424.779,Z 909.245,A -85,B 0,C 180,E1 -5821.609,E2 -5821.609} C_VEL
LIN {X 0,Y 422.704,Z 926.655,A -85,B 0,C 180,E1 -5823.898,E2 -5823.898} C_VEL
LIN {X 0,Y 420.882,Z 942.313,A -85,B 0,C 180,E1 -5826.329,E2 -5826.329} C_VEL
LIN {X 0,Y 419.26,Z 956.971,A -85,B 0,C 180,E1 -5829.039,E2 -5829.039} C_VEL
LIN {X 0,Y 417.98,Z 969.711,A -85,B 0,C 180,E1 -5831.882,E2 -5831.882} C_VEL
LIN {X 0,Y 417.129,Z 979.587,A -85,B 0,C 180,E1 -5834.569,E2 -5834.569} C_VEL
LIN {X 0,Y 416.563,Z 987.669,A -85,B 0,C 180,E1 -5837.242,E2 -5837.242} C_VEL
LIN {X 0,Y 416.185,Z 994.607,A -85,B 0,C 180,E1 -5840.178,E2 -5840.178} C_VEL
LIN {X 0,Y 416.038,Z 999.454,A -85,B 0,C 180,E1 -5843.002,E2 -5843.002} C_VEL
LIN {X 0,Y 415.989,Z 1002.612,A -85,B 0,C 180,E1 -5845.726,E2 -5845.726} C_VEL
LIN {X 0,Y 415.967,Z 1004.165,A -85,B 0,C 180,E1 -5848.484,E2 -5848.484} C_VEL
LIN {X 0,Y 415.969,Z 1004.359,A -85,B 0,C 180,E1 -5851.101,E2 -5851.101} C_VEL
LIN {X 0,Y 415.98,Z 1002.829,A -85,B 0,C 180,E1 -5854.055,E2 -5854.055} C_VEL
LIN {X 0,Y 416.022,Z 999.729,A -85,B 0,C 180,E1 -5856.901,E2 -5856.901} C_VEL
LIN {X 0,Y 416.164,Z 994.857,A -85,B 0,C 180,E1 -5859.821,E2 -5859.821} C_VEL
LIN {X 0,Y 416.528,Z 988.122,A -85,B 0,C 180,E1 -5862.758,E2 -5862.758} C_VEL
LIN {X 0,Y 417.131,Z 979.897,A -85,B 0,C 180,E1 -5865.572,E2 -5865.572} C_VEL
LIN {X 0,Y 418.059,Z 969.74,A -85,B 0,C 180,E1 -5868.403,E2 -5868.403} C_VEL
LIN {X 0,Y 419.403,Z 957.489,A -85,B 0,C 180,E1 -5871.229,E2 -5871.229} C_VEL
LIN {X 0,Y 421.147,Z 943.401,A -85,B 0,C 180,E1 -5873.952,E2 -5873.952} C_VEL
LIN {X 0,Y 423.255,Z 927.685,A -85,B 0,C 180,E1 -5876.517,E2 -5876.517} C_VEL
LIN {X 0,Y 425.707,Z 910.186,A -85,B 0,C 180,E1 -5878.936,E2 -5878.936} C_VEL
LIN {X 0,Y 428.261,Z 892.066,A -85,B 0,C 180,E1 -5881.062,E2 -5881.062} C_VEL
LIN {X 0,Y 430.842,Z 873.635,A -85,B 0,C 180,E1 -5882.891,E2 -5882.891} C_VEL
LIN {X 0,Y 433.595,Z 852.824,A -85,B 0,C 180,E1 -5884.64,E2 -5884.64} C_VEL
LIN {X 0,Y 436.111,Z 833.3,A -85,B 0,C 180,E1 -5886.012,E2 -5886.012} C_VEL
LIN {X 0,Y 438.475,Z 812.119,A -85,B 0,C 180,E1 -5887.222,E2 -5887.222} C_VEL
LIN {X 0,Y 440.732,Z 789.522,A -85,B 0,C 180,E1 -5888.247,E2 -5888.247} C_VEL
LIN {X 0,Y 442.589,Z 767.883,A -85,B 0,C 180,E1 -5888.993,E2 -5888.993} C_VEL
LIN {X 0,Y 443.885,Z 745.189,A -85,B 0,C 180,E1 -5889.54,E2 -5889.54} C_VEL
LIN {X 0,Y 445.112,Z 716.957,A -85,B 0,C 180,E1 -5890.053,E2 -5890.053} C_VEL
LIN {X 0,Y 445.481,Z 713.394,A -85,B 0,C 180,E1 -5890.102,E2 -5890.102} C_VEL
LIN {X 0,Y 451.204,Z 696.033,A -85,B 0,C 180,E1 -5890.919,E2 -5890.919} C_VEL
LIN {X 0,Y 458.598,Z 676.118,A -85,B 0,C 180,E1 -5891.764,E2 -5891.764} C_VEL
LIN {X 0,Y 466.972,Z 657.453,A -85,B 0,C 180,E1 -5892.412,E2 -5892.412} C_VEL
LIN {X 0,Y 474.756,Z 639.579,A -85,B 0,C 180,E1 -5893.028,E2 -5893.028} C_VEL
LIN {X 0,Y 485.781,Z 618.357,A -85,B 0,C 180,E1 -5893.573,E2 -5893.573} C_VEL
LIN {X 0,Y 496.752,Z 599.202,A -85,B 0,C 180,E1 -5893.954,E2 -5893.954} C_VEL
LIN {X 0,Y 486.854,Z 590.259,A -85,B 0,C 180,E1 -5895.548,E2 -5895.548} C_VEL
LIN {X 0,Y 477.876,Z 579.047,A -85,B 0,C 180,E1 -5897.32,E2 -5897.32} C_VEL
LIN {X 0,Y 471.079,Z 567.028,A -85,B 0,C 180,E1 -5899.016,E2 -5899.016} C_VEL
LIN {X 0,Y 465.849,Z 553.606,A -85,B 0,C 180,E1 -5900.717,E2 -5900.717} C_VEL
LIN {X 0,Y 462.311,Z 538.65,A -85,B 0,C 180,E1 -5902.419,E2 -5902.419} C_VEL
LIN {X 0,Y 460.532,Z 522.148,A -85,B 0,C 180,E1 -5904.113,E2 -5904.113} C_VEL
LIN {X 0,Y 460.401,Z 504.081,A -85,B 0,C 180,E1 -5905.773,E2 -5905.773} C_VEL
LIN {X 0,Y 462.441,Z 481.13,A -85,B 0,C 180,E1 -5907.655,E2 -5907.655} C_VEL
LIN {X 0,Y 464.709,Z 463.14,A -85,B 0,C 180,E1 -5909.055,E2 -5909.055} C_VEL
LIN {X 0,Y 455.383,Z 445.713,A -85,B 0,C 180,E1 -5912.259,E2 -5912.259} C_VEL
LIN {X 0,Y 447.582,Z 431.653,A -85,B 0,C 180,E1 -5915.089,E2 -5915.089} C_VEL
LIN {X 0,Y 440.097,Z 418.351,A -85,B 0,C 180,E1 -5917.962,E2 -5917.962} C_VEL
LIN {X 0,Y 434.473,Z 408.686,A -85,B 0,C 180,E1 -5920.228,E2 -5920.228} C_VEL
LIN {X 0,Y 431.466,Z 403.55,A -85,B 0,C 180,E1 -5921.49,E2 -5921.49} C_VEL
LIN {X 0,Y 428.488,Z 398.447,A -85,B 0,C 180,E1 -5922.762,E2 -5922.762} C_VEL
LIN {X 0,Y 425.958,Z 393.942,A -85,B 0,C 180,E1 -5923.92,E2 -5923.92} C_VEL
LIN {X 0,Y 423.659,Z 389.994,A -85,B 0,C 180,E1 -5924.954,E2 -5924.954} C_VEL
LIN {X 0,Y 420.806,Z 385.407,A -85,B 0,C 180,E1 -5926.255,E2 -5926.255} C_VEL
LIN {X 0,Y 420.065,Z 383.786,A -85,B 0,C 180,E1 -5926.651,E2 -5926.651} C_VEL
LIN {X 0,Y 417.921,Z 380.912,A -85,B 0,C 180,E1 -5927.566,E2 -5927.566} C_VEL
LIN {X 0,Y 417.346,Z 378.745,A -85,B 0,C 180,E1 -5928.067,E2 -5928.067} C_VEL
LIN {X 0,Y 417.376,Z 378.743,A -85,B 0,C 180,E1 -5931.875,E2 -5931.875} C_VEL
LIN {X 0,Y 417.335,Z 378.752,A -85,B 0,C 180,E1 -5935.741,E2 -5935.741} C_VEL
LIN {X 0,Y 417.383,Z 378.751,A -85,B 0,C 180,E1 -5939.589,E2 -5939.589} C_VEL
LIN {X 0,Y 417.35,Z 378.752,A -85,B 0,C 180,E1 -5943.434,E2 -5943.434} C_VEL
LIN {X 0,Y 417.388,Z 378.746,A -85,B 0,C 180,E1 -5947.294,E2 -5947.294} C_VEL
LIN {X 0,Y 417.369,Z 378.749,A -85,B 0,C 180,E1 -5951.189,E2 -5951.189} C_VEL
LIN {X 0,Y 417.367,Z 378.743,A -85,B 0,C 180,E1 -5954.995,E2 -5954.995} C_VEL
LIN {X 0,Y 417.353,Z 378.746,A -85,B 0,C 180,E1 -5959.015,E2 -5959.015} C_VEL
LIN {X 0,Y 417.371,Z 378.746,A -85,B 0,C 180,E1 -5962.734,E2 -5962.734} C_VEL
LIN {X 0,Y 417.343,Z 378.741,A -85,B 0,C 180,E1 -5966.77,E2 -5966.77} C_VEL
LIN {X 0,Y 417.383,Z 378.738,A -85,B 0,C 180,E1 -5970.521,E2 -5970.521} C_VEL
LIN {X 0,Y 417.357,Z 378.736,A -85,B 0,C 180,E1 -5974.501,E2 -5974.501} C_VEL
LIN {X 0,Y 417.383,Z 378.727,A -85,B 0,C 180,E1 -5978.349,E2 -5978.349} C_VEL
LIN {X 0,Y 417.377,Z 378.712,A -85,B 0,C 180,E1 -5982.312,E2 -5982.312} C_VEL
LIN {X 0,Y 417.359,Z 378.731,A -85,B 0,C 180,E1 -5986.146,E2 -5986.146} C_VEL
LIN {X 0,Y 417.396,Z 378.87,A -85,B 0,C 180,E1 -5986.583,E2 -5986.583} C_VEL
LIN {X 0,Y 418.504,Z 381.953,A -85,B 0,C 180,E1 -5986.977,E2 -5986.977} C_VEL
LIN {X 0,Y 423.126,Z 391.208,A -85,B 0,C 180,E1 -5988.307,E2 -5988.307} C_VEL
LIN {X 0,Y 431.094,Z 409.46,A -85,B 0,C 180,E1 -5990.775,E2 -5990.775} C_VEL
LIN {X 0,Y 438.283,Z 428.761,A -85,B 0,C 180,E1 -5993.201,E2 -5993.201} C_VEL
LIN {X 0,Y 436.233,Z 472.575,A -85,B 0,C 180,E1 -5996.627,E2 -5996.627} C_VEL
LIN {X 0,Y 435.833,Z 493.055,A -85,B 0,C 180,E1 -5998.075,E2 -5998.075} C_VEL
LIN {X 0,Y 436.795,Z 501.218,A -85,B 0,C 180,E1 -5998.314,E2 -5998.314} C_VEL
LIN {X 0,Y 432.861,Z 683.769,A -85,B 0,C 180,E1 -6001.462,E2 -6001.462} C_VEL
LIN {X 0,Y 431.873,Z 691.46,A -85,B 0,C 180,E1 -6001.531,E2 -6001.531} C_VEL
LIN {X 0,Y 426.579,Z 709.698,A -85,B 0,C 180,E1 -6001.584,E2 -6001.584} C_VEL
LIN {X 0,Y 425.314,Z 716.154,A -85,B 0,C 180,E1 -6001.705,E2 -6001.705} C_VEL
LIN {X 0,Y 425.206,Z 718.299,A -85,B 0,C 180,E1 -6001.782,E2 -6001.782} C_VEL
LIN {X 0,Y 424.31,Z 736.654,A -85,B 0,C 180,E1 -6002.569,E2 -6002.569} C_VEL
LIN {X 0,Y 423.082,Z 753.695,A -85,B 0,C 180,E1 -6003.547,E2 -6003.547} C_VEL
LIN {X 0,Y 421.517,Z 770.785,A -85,B 0,C 180,E1 -6004.8,E2 -6004.8} C_VEL
LIN {X 0,Y 419.807,Z 786.75,A -85,B 0,C 180,E1 -6006.265,E2 -6006.265} C_VEL
LIN {X 0,Y 418.031,Z 801.06,A -85,B 0,C 180,E1 -6007.87,E2 -6007.87} C_VEL
LIN {X 0,Y 416.302,Z 813.979,A -85,B 0,C 180,E1 -6009.62,E2 -6009.62} C_VEL
LIN {X 0,Y 414.615,Z 826.032,A -85,B 0,C 180,E1 -6011.585,E2 -6011.585} C_VEL
LIN {X 0,Y 413.09,Z 836.718,A -85,B 0,C 180,E1 -6013.694,E2 -6013.694} C_VEL
LIN {X 0,Y 411.805,Z 846.053,A -85,B 0,C 180,E1 -6015.949,E2 -6015.949} C_VEL
LIN {X 0,Y 410.763,Z 854.012,A -85,B 0,C 180,E1 -6018.344,E2 -6018.344} C_VEL
LIN {X 0,Y 409.989,Z 860.54,A -85,B 0,C 180,E1 -6020.879,E2 -6020.879} C_VEL
LIN {X 0,Y 409.495,Z 865.542,A -85,B 0,C 180,E1 -6023.551,E2 -6023.551} C_VEL
LIN {X 0,Y 409.219,Z 868.74,A -85,B 0,C 180,E1 -6026.218,E2 -6026.218} C_VEL
LIN {X 0,Y 409.092,Z 870.263,A -85,B 0,C 180,E1 -6028.88,E2 -6028.88} C_VEL
LIN {X 0,Y 409.105,Z 870.127,A -85,B 0,C 180,E1 -6031.605,E2 -6031.605} C_VEL
LIN {X 0,Y 409.247,Z 868.417,A -85,B 0,C 180,E1 -6034.204,E2 -6034.204} C_VEL
LIN {X 0,Y 409.537,Z 864.992,A -85,B 0,C 180,E1 -6036.871,E2 -6036.871} C_VEL
LIN {X 0,Y 410.037,Z 860.096,A -85,B 0,C 180,E1 -6039.403,E2 -6039.403} C_VEL
LIN {X 0,Y 410.837,Z 853.427,A -85,B 0,C 180,E1 -6041.942,E2 -6041.942} C_VEL
LIN {X 0,Y 411.976,Z 844.791,A -85,B 0,C 180,E1 -6044.477,E2 -6044.477} C_VEL
LIN {X 0,Y 413.313,Z 835.166,A -85,B 0,C 180,E1 -6046.731,E2 -6046.731} C_VEL
LIN {X 0,Y 414.891,Z 824.15,A -85,B 0,C 180,E1 -6048.841,E2 -6048.841} C_VEL
LIN {X 0,Y 416.622,Z 811.714,A -85,B 0,C 180,E1 -6050.805,E2 -6050.805} C_VEL
LIN {X 0,Y 418.474,Z 797.75,A -85,B 0,C 180,E1 -6052.624,E2 -6052.624} C_VEL
LIN {X 0,Y 420.289,Z 782.738,A -85,B 0,C 180,E1 -6054.229,E2 -6054.229} C_VEL
LIN {X 0,Y 421.937,Z 766.727,A -85,B 0,C 180,E1 -6055.625,E2 -6055.625} C_VEL
LIN {X 0,Y 423.453,Z 749.67,A -85,B 0,C 180,E1 -6056.808,E2 -6056.808} C_VEL
LIN {X 0,Y 424.611,Z 732.071,A -85,B 0,C 180,E1 -6057.753,E2 -6057.753} C_VEL
LIN {X 0,Y 425.417,Z 713.347,A -85,B 0,C 180,E1 -6058.484,E2 -6058.484} C_VEL
LIN {X 0,Y 425.793,Z 694.043,A -85,B 0,C 180,E1 -6058.978,E2 -6058.978} C_VEL
LIN {X 0,Y 429.947,Z 499.818,A -85,B 0,C 180,E1 -6062.399,E2 -6062.399} C_VEL
LIN {X 0,Y 429.046,Z 492.932,A -85,B 0,C 180,E1 -6062.65,E2 -6062.65} C_VEL
LIN {X 0,Y 430.16,Z 459.347,A -85,B 0,C 180,E1 -6065.144,E2 -6065.144} C_VEL
LIN {X 0,Y 431.478,Z 431.682,A -85,B 0,C 180,E1 -6067.36,E2 -6067.36} C_VEL
LIN {X 0,Y 424.322,Z 412.613,A -85,B 0,C 180,E1 -6069.809,E2 -6069.809} C_VEL
LIN {X 0,Y 416.757,Z 395.273,A -85,B 0,C 180,E1 -6072.204,E2 -6072.204} C_VEL
LIN {X 0,Y 414.182,Z 390.401,A -85,B 0,C 180,E1 -6072.975,E2 -6072.975} C_VEL
LIN {X 0,Y 420.657,Z 404.308,A -85,B 0,C 180,E1 -6075.486,E2 -6075.486} C_VEL
LIN {X 0,Y 428.034,Z 421.793,A -85,B 0,C 180,E1 -6078.375,E2 -6078.375} C_VEL
LIN {X 0,Y 434.538,Z 438.825,A -85,B 0,C 180,E1 -6080.958,E2 -6080.958} C_VEL
LIN {X 0,Y 430.732,Z 478.854,A -85,B 0,C 180,E1 -6084.689,E2 -6084.689} C_VEL
LIN {X 0,Y 426.941,Z 522.234,A -85,B 0,C 180,E1 -6088.674,E2 -6088.674} C_VEL
LIN {X 0,Y 423.36,Z 567.905,A -85,B 0,C 180,E1 -6092.806,E2 -6092.806} C_VEL
LIN {X 0,Y 421.002,Z 602.971,A -85,B 0,C 180,E1 -6095.906,E2 -6095.906} C_VEL
LIN {X 0,Y 421.752,Z 611.795,A -85,B 0,C 180,E1 -6096.181,E2 -6096.181} C_VEL
LIN {X 0,Y 417.16,Z 749.337,A -85,B 0,C 180,E1 -6099.351,E2 -6099.351} C_VEL
LIN {X 0,Y 416.644,Z 766.336,A -85,B 0,C 180,E1 -6100.003,E2 -6100.003} C_VEL
LIN {X 0,Y 415.93,Z 781.836,A -85,B 0,C 180,E1 -6100.844,E2 -6100.844} C_VEL
LIN {X 0,Y 415.008,Z 797.293,A -85,B 0,C 180,E1 -6101.965,E2 -6101.965} C_VEL
LIN {X 0,Y 414.065,Z 810.735,A -85,B 0,C 180,E1 -6103.197,E2 -6103.197} C_VEL
LIN {X 0,Y 413,Z 824.38,A -85,B 0,C 180,E1 -6104.771,E2 -6104.771} C_VEL
LIN {X 0,Y 412.079,Z 835.746,A -85,B 0,C 180,E1 -6106.387,E2 -6106.387} C_VEL
LIN {X 0,Y 411.235,Z 846.085,A -85,B 0,C 180,E1 -6108.215,E2 -6108.215} C_VEL
LIN {X 0,Y 410.552,Z 855.047,A -85,B 0,C 180,E1 -6110.184,E2 -6110.184} C_VEL
LIN {X 0,Y 410.031,Z 862.484,A -85,B 0,C 180,E1 -6112.292,E2 -6112.292} C_VEL
LIN {X 0,Y 409.704,Z 868.424,A -85,B 0,C 180,E1 -6114.538,E2 -6114.538} C_VEL
LIN {X 0,Y 409.556,Z 872.418,A -85,B 0,C 180,E1 -6116.781,E2 -6116.781} C_VEL
LIN {X 0,Y 409.557,Z 874.742,A -85,B 0,C 180,E1 -6119.02,E2 -6119.02} C_VEL
LIN {X 0,Y 409.682,Z 875.341,A -85,B 0,C 180,E1 -6121.258,E2 -6121.258} C_VEL
LIN {X 0,Y 409.955,Z 874.192,A -85,B 0,C 180,E1 -6123.635,E2 -6123.635} C_VEL
LIN {X 0,Y 410.392,Z 871.319,A -85,B 0,C 180,E1 -6125.873,E2 -6125.873} C_VEL
LIN {X 0,Y 411.054,Z 866.696,A -85,B 0,C 180,E1 -6128.11,E2 -6128.11} C_VEL
LIN {X 0,Y 411.903,Z 860.483,A -85,B 0,C 180,E1 -6130.206,E2 -6130.206} C_VEL
LIN {X 0,Y 412.928,Z 852.956,A -85,B 0,C 180,E1 -6132.161,E2 -6132.161} C_VEL
LIN {X 0,Y 414.084,Z 844.018,A -85,B 0,C 180,E1 -6133.972,E2 -6133.972} C_VEL
LIN {X 0,Y 415.465,Z 832.877,A -85,B 0,C 180,E1 -6135.78,E2 -6135.78} C_VEL
LIN {X 0,Y 416.917,Z 819.843,A -85,B 0,C 180,E1 -6137.444,E2 -6137.444} C_VEL
LIN {X 0,Y 418.148,Z 806.866,A -85,B 0,C 180,E1 -6138.754,E2 -6138.754} C_VEL
LIN {X 0,Y 419.25,Z 793.08,A -85,B 0,C 180,E1 -6139.867,E2 -6139.867} C_VEL
LIN {X 0,Y 420.115,Z 778.42,A -85,B 0,C 180,E1 -6140.769,E2 -6140.769} C_VEL
LIN {X 0,Y 420.764,Z 762.393,A -85,B 0,C 180,E1 -6141.502,E2 -6141.502} C_VEL
LIN {X 0,Y 422.954,Z 731.392,A -85,B 0,C 180,E1 -6142.678,E2 -6142.678} C_VEL
LIN {X 0,Y 434.605,Z 634.358,A -85,B 0,C 180,E1 -6146.176,E2 -6146.176} C_VEL
LIN {X 0,Y 439.674,Z 621.705,A -85,B 0,C 180,E1 -6147.053,E2 -6147.053} C_VEL
LIN {X 0,Y 447.183,Z 592.885,A -85,B 0,C 180,E1 -6150.278,E2 -6150.278} C_VEL
LIN {X 0,Y 455.275,Z 570.049,A -85,B 0,C 180,E1 -6153,E2 -6153} C_VEL
LIN {X 0,Y 463.475,Z 553.013,A -85,B 0,C 180,E1 -6155.169,E2 -6155.169} C_VEL
LIN {X 0,Y 467.756,Z 545.854,A -85,B 0,C 180,E1 -6156.113,E2 -6156.113} C_VEL
LIN {X 0,Y 464.061,Z 554.185,A -85,B 0,C 180,E1 -6157.745,E2 -6157.745} C_VEL
LIN {X 0,Y 462.794,Z 562.201,A -85,B 0,C 180,E1 -6159.334,E2 -6159.334} C_VEL
LIN {X 0,Y 463.769,Z 570.432,A -85,B 0,C 180,E1 -6160.95,E2 -6160.95} C_VEL
LIN {X 0,Y 467.034,Z 578.943,A -85,B 0,C 180,E1 -6162.571,E2 -6162.571} C_VEL
LIN {X 0,Y 472.958,Z 587.906,A -85,B 0,C 180,E1 -6164.237,E2 -6164.237} C_VEL
LIN {X 0,Y 480.517,Z 596.044,A -85,B 0,C 180,E1 -6165.708,E2 -6165.708} C_VEL
LIN {X 0,Y 483.86,Z 599.152,A -85,B 0,C 180,E1 -6166.246,E2 -6166.246} C_VEL
LIN {X 0,Y 470.795,Z 622.479,A -85,B 0,C 180,E1 -6166.756,E2 -6166.756} C_VEL
LIN {X 0,Y 461.166,Z 642.374,A -85,B 0,C 180,E1 -6167.348,E2 -6167.348} C_VEL
LIN {X 0,Y 454.437,Z 658.411,A -85,B 0,C 180,E1 -6167.935,E2 -6167.935} C_VEL
LIN {X 0,Y 446.641,Z 676.378,A -85,B 0,C 180,E1 -6168.576,E2 -6168.576} C_VEL
LIN {X 0,Y 437.156,Z 703.955,A -85,B 0,C 180,E1 -6169.786,E2 -6169.786} C_VEL
LIN {X 0,Y 434.965,Z 725.185,A -85,B 0,C 180,E1 -6170.108,E2 -6170.108} C_VEL
LIN {X 0,Y 433.546,Z 753.364,A -85,B 0,C 180,E1 -6170.769,E2 -6170.769} C_VEL
LIN {X 0,Y 431.399,Z 779.265,A -85,B 0,C 180,E1 -6171.621,E2 -6171.621} C_VEL
LIN {X 0,Y 429.245,Z 802.562,A -85,B 0,C 180,E1 -6172.641,E2 -6172.641} C_VEL
LIN {X 0,Y 426.857,Z 825.477,A -85,B 0,C 180,E1 -6173.912,E2 -6173.912} C_VEL
LIN {X 0,Y 424.28,Z 848.542,A -85,B 0,C 180,E1 -6175.475,E2 -6175.475} C_VEL
LIN {X 0,Y 421.825,Z 869.775,A -85,B 0,C 180,E1 -6177.206,E2 -6177.206} C_VEL
LIN {X 0,Y 419.347,Z 889.916,A -85,B 0,C 180,E1 -6179.16,E2 -6179.16} C_VEL
LIN {X 0,Y 417.062,Z 908.395,A -85,B 0,C 180,E1 -6181.27,E2 -6181.27} C_VEL
LIN {X 0,Y 414.967,Z 925.278,A -85,B 0,C 180,E1 -6183.528,E2 -6183.528} C_VEL
LIN {X 0,Y 413.067,Z 941.03,A -85,B 0,C 180,E1 -6186.005,E2 -6186.005} C_VEL
LIN {X 0,Y 411.382,Z 955.78,A -85,B 0,C 180,E1 -6188.768,E2 -6188.768} C_VEL
LIN {X 0,Y 410.06,Z 968.597,A -85,B 0,C 180,E1 -6191.666,E2 -6191.666} C_VEL
LIN {X 0,Y 409.15,Z 979.017,A -85,B 0,C 180,E1 -6194.551,E2 -6194.551} C_VEL
LIN {X 0,Y 408.596,Z 986.97,A -85,B 0,C 180,E1 -6197.277,E2 -6197.277} C_VEL
LIN {X 0,Y 408.242,Z 993.573,A -85,B 0,C 180,E1 -6200.128,E2 -6200.128} C_VEL
LIN {X 0,Y 408.103,Z 998.561,A -85,B 0,C 180,E1 -6203.105,E2 -6203.105} C_VEL
LIN {X 0,Y 408.061,Z 1001.67,A -85,B 0,C 180,E1 -6205.925,E2 -6205.925} C_VEL
LIN {X 0,Y 408.047,Z 1003.115,A -85,B 0,C 180,E1 -6208.736,E2 -6208.736} C_VEL
LIN {X 0,Y 408.044,Z 1003.162,A -85,B 0,C 180,E1 -6211.404,E2 -6211.404} C_VEL
LIN {X 0,Y 408.048,Z 1001.563,A -85,B 0,C 180,E1 -6214.356,E2 -6214.356} C_VEL
LIN {X 0,Y 408.07,Z 998.415,A -85,B 0,C 180,E1 -6217.178,E2 -6217.178} C_VEL
LIN {X 0,Y 408.221,Z 993.618,A -85,B 0,C 180,E1 -6220.064,E2 -6220.064} C_VEL
LIN {X 0,Y 408.606,Z 986.669,A -85,B 0,C 180,E1 -6223.12,E2 -6223.12} C_VEL
LIN {X 0,Y 409.298,Z 977.74,A -85,B 0,C 180,E1 -6226.169,E2 -6226.169} C_VEL
LIN {X 0,Y 410.318,Z 967.299,A -85,B 0,C 180,E1 -6229.058,E2 -6229.058} C_VEL
LIN {X 0,Y 411.709,Z 955.342,A -85,B 0,C 180,E1 -6231.812,E2 -6231.812} C_VEL
LIN {X 0,Y 413.468,Z 941.923,A -85,B 0,C 180,E1 -6234.426,E2 -6234.426} C_VEL
LIN {X 0,Y 415.708,Z 926.097,A -85,B 0,C 180,E1 -6237.038,E2 -6237.038} C_VEL
LIN {X 0,Y 418.221,Z 909.07,A -85,B 0,C 180,E1 -6239.421,E2 -6239.421} C_VEL
LIN {X 0,Y 420.931,Z 890.879,A -85,B 0,C 180,E1 -6241.585,E2 -6241.585} C_VEL
LIN {X 0,Y 423.634,Z 872.371,A -85,B 0,C 180,E1 -6243.442,E2 -6243.442} C_VEL
LIN {X 0,Y 426.421,Z 852.38,A -85,B 0,C 180,E1 -6245.144,E2 -6245.144} C_VEL
LIN {X 0,Y 429.059,Z 832.844,A -85,B 0,C 180,E1 -6246.541,E2 -6246.541} C_VEL
LIN {X 0,Y 431.526,Z 811.941,A -85,B 0,C 180,E1 -6247.758,E2 -6247.758} C_VEL
LIN {X 0,Y 433.962,Z 788.791,A -85,B 0,C 180,E1 -6248.824,E2 -6248.824} C_VEL
LIN {X 0,Y 435.911,Z 767.03,A -85,B 0,C 180,E1 -6249.583,E2 -6249.583} C_VEL
LIN {X 0,Y 437.263,Z 744.377,A -85,B 0,C 180,E1 -6250.136,E2 -6250.136} C_VEL
LIN {X 0,Y 438.564,Z 716.997,A -85,B 0,C 180,E1 -6250.649,E2 -6250.649} C_VEL
LIN {X 0,Y 439.094,Z 712.371,A -85,B 0,C 180,E1 -6250.721,E2 -6250.721} C_VEL
LIN {X 0,Y 444.853,Z 695.245,A -85,B 0,C 180,E1 -6251.532,E2 -6251.532} C_VEL
LIN {X 0,Y 452.368,Z 675.256,A -85,B 0,C 180,E1 -6252.387,E2 -6252.387} C_VEL
LIN {X 0,Y 460.798,Z 656.628,A -85,B 0,C 180,E1 -6253.032,E2 -6253.032} C_VEL
LIN {X 0,Y 468.549,Z 638.972,A -85,B 0,C 180,E1 -6253.648,E2 -6253.648} C_VEL
LIN {X 0,Y 479.171,Z 618.472,A -85,B 0,C 180,E1 -6254.182,E2 -6254.182} C_VEL
LIN {X 0,Y 488.154,Z 602.512,A -85,B 0,C 180,E1 -6254.512,E2 -6254.512} C_VEL
LIN {X 0,Y 478.88,Z 593.244,A -85,B 0,C 180,E1 -6256.118,E2 -6256.118} C_VEL
LIN {X 0,Y 470.187,Z 581.431,A -85,B 0,C 180,E1 -6257.945,E2 -6257.945} C_VEL
LIN {X 0,Y 463.294,Z 567.839,A -85,B 0,C 180,E1 -6259.813,E2 -6259.813} C_VEL
LIN {X 0,Y 458.523,Z 553.647,A -85,B 0,C 180,E1 -6261.577,E2 -6261.577} C_VEL
LIN {X 0,Y 455.494,Z 537.889,A -85,B 0,C 180,E1 -6263.34,E2 -6263.34} C_VEL
LIN {X 0,Y 454.172,Z 519.263,A -85,B 0,C 180,E1 -6265.201,E2 -6265.201} C_VEL
LIN {X 0,Y 454.791,Z 500.43,A -85,B 0,C 180,E1 -6266.89,E2 -6266.89} C_VEL
LIN {X 0,Y 458.636,Z 467.369,A -85,B 0,C 180,E1 -6269.545,E2 -6269.545} C_VEL
LIN {X 0,Y 448.863,Z 448.98,A -85,B 0,C 180,E1 -6272.973,E2 -6272.973} C_VEL
LIN {X 0,Y 439.475,Z 432.116,A -85,B 0,C 180,E1 -6276.472,E2 -6276.472} C_VEL
LIN {X 0,Y 432.076,Z 419.126,A -85,B 0,C 180,E1 -6279.407,E2 -6279.407} C_VEL
LIN {X 0,Y 426.594,Z 409.707,A -85,B 0,C 180,E1 -6281.696,E2 -6281.696} C_VEL
LIN {X 0,Y 423.322,Z 404.147,A -85,B 0,C 180,E1 -6283.111,E2 -6283.111} C_VEL
LIN {X 0,Y 420.72,Z 399.639,A -85,B 0,C 180,E1 -6284.281,E2 -6284.281} C_VEL
LIN {X 0,Y 417.895,Z 394.79,A -85,B 0,C 180,E1 -6285.592,E2 -6285.592} C_VEL
LIN {X 0,Y 415.684,Z 390.859,A -85,B 0,C 180,E1 -6286.65,E2 -6286.65} C_VEL
LIN {X 0,Y 412.867,Z 386.402,A -85,B 0,C 180,E1 -6287.979,E2 -6287.979} C_VEL
LIN {X 0,Y 412.151,Z 384.812,A -85,B 0,C 180,E1 -6288.384,E2 -6288.384} C_VEL
LIN {X 0,Y 410.035,Z 381.998,A -85,B 0,C 180,E1 -6289.32,E2 -6289.32} C_VEL
LIN {X 0,Y 409.423,Z 379.733,A -85,B 0,C 180,E1 -6289.873,E2 -6289.873} C_VEL
LIN {X 0,Y 409.416,Z 379.736,A -85,B 0,C 180,E1 -6293.697,E2 -6293.697} C_VEL
LIN {X 0,Y 409.421,Z 379.74,A -85,B 0,C 180,E1 -6297.761,E2 -6297.761} C_VEL
LIN {X 0,Y 409.426,Z 379.741,A -85,B 0,C 180,E1 -6301.54,E2 -6301.54} C_VEL
LIN {X 0,Y 409.428,Z 379.736,A -85,B 0,C 180,E1 -6305.606,E2 -6305.606} C_VEL
LIN {X 0,Y 409.435,Z 379.738,A -85,B 0,C 180,E1 -6309.417,E2 -6309.417} C_VEL
LIN {X 0,Y 409.445,Z 379.733,A -85,B 0,C 180,E1 -6313.415,E2 -6313.415} C_VEL
LIN {X 0,Y 409.417,Z 379.738,A -85,B 0,C 180,E1 -6317.278,E2 -6317.278} C_VEL
LIN {X 0,Y 409.441,Z 379.73,A -85,B 0,C 180,E1 -6321.188,E2 -6321.188} C_VEL
LIN {X 0,Y 409.4,Z 379.739,A -85,B 0,C 180,E1 -6325.148,E2 -6325.148} C_VEL
LIN {X 0,Y 409.443,Z 379.734,A -85,B 0,C 180,E1 -6329.076,E2 -6329.076} C_VEL
LIN {X 0,Y 409.399,Z 379.74,A -85,B 0,C 180,E1 -6332.999,E2 -6332.999} C_VEL
LIN {X 0,Y 409.433,Z 379.692,A -85,B 0,C 180,E1 -6337.008,E2 -6337.008} C_VEL
LIN {X 0,Y 409.404,Z 379.724,A -85,B 0,C 180,E1 -6340.792,E2 -6340.792} C_VEL
LIN {X 0,Y 409.443,Z 379.738,A -85,B 0,C 180,E1 -6344.715,E2 -6344.715} C_VEL
LIN {X 0,Y 409.441,Z 379.879,A -85,B 0,C 180,E1 -6345.666,E2 -6345.666} C_VEL
LIN {X 0,Y 410.686,Z 383.145,A -85,B 0,C 180,E1 -6346.108,E2 -6346.108} C_VEL
LIN {X 0,Y 411.724,Z 384.936,A -85,B 0,C 180,E1 -6346.395,E2 -6346.395} C_VEL
LIN {X 0,Y 420.395,Z 403.269,A -85,B 0,C 180,E1 -6349.038,E2 -6349.038} C_VEL
LIN {X 0,Y 427.714,Z 421.348,A -85,B 0,C 180,E1 -6351.44,E2 -6351.44} C_VEL
LIN {X 0,Y 431.543,Z 432.144,A -85,B 0,C 180,E1 -6352.792,E2 -6352.792} C_VEL
LIN {X 0,Y 429.508,Z 474.518,A -85,B 0,C 180,E1 -6356.115,E2 -6356.115} C_VEL
LIN {X 0,Y 429.116,Z 494.342,A -85,B 0,C 180,E1 -6357.517,E2 -6357.517} C_VEL
LIN {X 0,Y 430.048,Z 502.367,A -85,B 0,C 180,E1 -6357.757,E2 -6357.757} C_VEL
LIN {X 0,Y 425.682,Z 700.753,A -85,B 0,C 180,E1 -6361.264,E2 -6361.264} C_VEL
LIN {X 0,Y 425.206,Z 718.299,A -85,B 0,C 180,E1 -6361.782,E2 -6361.782} C_VEL
LIN {X 0,Y 424.032,Z 725.845,A -85,B 0,C 180,E1 -6362.001,E2 -6362.001} C_VEL
LIN {X 0,Y 418.084,Z 743.561,A -85,B 0,C 180,E1 -6362.448,E2 -6362.448} C_VEL
LIN {X 0,Y 416.429,Z 750.708,A -85,B 0,C 180,E1 -6362.788,E2 -6362.788} C_VEL
LIN {X 0,Y 416.316,Z 751.71,A -85,B 0,C 180,E1 -6362.851,E2 -6362.851} C_VEL
LIN {X 0,Y 414.721,Z 768.743,A -85,B 0,C 180,E1 -6364.063,E2 -6364.063} C_VEL
LIN {X 0,Y 413.009,Z 784.501,A -85,B 0,C 180,E1 -6365.469,E2 -6365.469} C_VEL
LIN {X 0,Y 411.112,Z 799.423,A -85,B 0,C 180,E1 -6367.1,E2 -6367.1} C_VEL
LIN {X 0,Y 409.167,Z 813.316,A -85,B 0,C 180,E1 -6368.948,E2 -6368.948} C_VEL
LIN {X 0,Y 407.226,Z 826.495,A -85,B 0,C 180,E1 -6371.089,E2 -6371.089} C_VEL
LIN {X 0,Y 405.587,Z 837.323,A -85,B 0,C 180,E1 -6373.236,E2 -6373.236} C_VEL
LIN {X 0,Y 404.195,Z 846.781,A -85,B 0,C 180,E1 -6375.532,E2 -6375.532} C_VEL
LIN {X 0,Y 403.061,Z 854.85,A -85,B 0,C 180,E1 -6377.973,E2 -6377.973} C_VEL
LIN {X 0,Y 402.207,Z 861.477,A -85,B 0,C 180,E1 -6380.557,E2 -6380.557} C_VEL
LIN {X 0,Y 401.672,Z 866.338,A -85,B 0,C 180,E1 -6383.138,E2 -6383.138} C_VEL
LIN {X 0,Y 401.357,Z 869.729,A -85,B 0,C 180,E1 -6385.857,E2 -6385.857} C_VEL
LIN {X 0,Y 401.206,Z 871.44,A -85,B 0,C 180,E1 -6388.572,E2 -6388.572} C_VEL
LIN {X 0,Y 401.196,Z 871.52,A -85,B 0,C 180,E1 -6391.286,E2 -6391.286} C_VEL
LIN {X 0,Y 401.341,Z 869.967,A -85,B 0,C 180,E1 -6394,E2 -6394} C_VEL
LIN {X 0,Y 401.642,Z 866.728,A -85,B 0,C 180,E1 -6396.72,E2 -6396.72} C_VEL
LIN {X 0,Y 402.188,Z 861.689,A -85,B 0,C 180,E1 -6399.444,E2 -6399.444} C_VEL
LIN {X 0,Y 403.029,Z 855.128,A -85,B 0,C 180,E1 -6402.029,E2 -6402.029} C_VEL
LIN {X 0,Y 404.153,Z 847.13,A -85,B 0,C 180,E1 -6404.47,E2 -6404.47} C_VEL
LIN {X 0,Y 405.533,Z 837.748,A -85,B 0,C 180,E1 -6406.767,E2 -6406.767} C_VEL
LIN {X 0,Y 407.163,Z 827.007,A -85,B 0,C 180,E1 -6408.914,E2 -6408.914} C_VEL
LIN {X 0,Y 408.993,Z 814.629,A -85,B 0,C 180,E1 -6410.953,E2 -6410.953} C_VEL
LIN {X 0,Y 410.944,Z 800.735,A -85,B 0,C 180,E1 -6412.835,E2 -6412.835} C_VEL
LIN {X 0,Y 412.829,Z 786.083,A -85,B 0,C 180,E1 -6414.467,E2 -6414.467} C_VEL
LIN {X 0,Y 414.563,Z 770.45,A -85,B 0,C 180,E1 -6415.892,E2 -6415.892} C_VEL
LIN {X 0,Y 416.114,Z 754.13,A -85,B 0,C 180,E1 -6417.087,E2 -6417.087} C_VEL
LIN {X 0,Y 417.394,Z 736.815,A -85,B 0,C 180,E1 -6418.081,E2 -6418.081} C_VEL
LIN {X 0,Y 418.31,Z 718.452,A -85,B 0,C 180,E1 -6418.866,E2 -6418.866} C_VEL
LIN {X 0,Y 418.798,Z 699.98,A -85,B 0,C 180,E1 -6419.4,E2 -6419.4} C_VEL
LIN {X 0,Y 423.252,Z 501.051,A -85,B 0,C 180,E1 -6422.973,E2 -6422.973} C_VEL
LIN {X 0,Y 422.369,Z 494.111,A -85,B 0,C 180,E1 -6423.232,E2 -6423.232} C_VEL
LIN {X 0,Y 423.549,Z 460.479,A -85,B 0,C 180,E1 -6425.743,E2 -6425.743} C_VEL
LIN {X 0,Y 424.919,Z 435.341,A -85,B 0,C 180,E1 -6427.755,E2 -6427.755} C_VEL
LIN {X 0,Y 417.669,Z 416.1,A -85,B 0,C 180,E1 -6430.268,E2 -6430.268} C_VEL
LIN {X 0,Y 410.852,Z 400.267,A -85,B 0,C 180,E1 -6432.49,E2 -6432.49} C_VEL
LIN {X 0,Y 409.044,Z 396.988,A -85,B 0,C 180,E1 -6433.015,E2 -6433.015} C_VEL
LIN {X 0,Y 416.441,Z 413.475,A -85,B 0,C 180,E1 -6435.98,E2 -6435.98} C_VEL
LIN {X 0,Y 423.812,Z 431.424,A -85,B 0,C 180,E1 -6438.918,E2 -6438.918} C_VEL
LIN {X 0,Y 427.742,Z 442.232,A -85,B 0,C 180,E1 -6440.563,E2 -6440.563} C_VEL
LIN {X 0,Y 423.695,Z 483.377,A -85,B 0,C 180,E1 -6444.429,E2 -6444.429} C_VEL
LIN {X 0,Y 419.646,Z 527.756,A -85,B 0,C 180,E1 -6448.547,E2 -6448.547} C_VEL
LIN {X 0,Y 415.871,Z 573.974,A -85,B 0,C 180,E1 -6452.77,E2 -6452.77} C_VEL
LIN {X 0,Y 413.792,Z 603.774,A -85,B 0,C 180,E1 -6455.43,E2 -6455.43} C_VEL
LIN {X 0,Y 414.54,Z 612.758,A -85,B 0,C 180,E1 -6455.717,E2 -6455.717} C_VEL
LIN {X 0,Y 409.649,Z 749.904,A -85,B 0,C 180,E1 -6458.977,E2 -6458.977} C_VEL
LIN {X 0,Y 409.095,Z 767.253,A -85,B 0,C 180,E1 -6459.655,E2 -6459.655} C_VEL
LIN {X 0,Y 408.315,Z 783.279,A -85,B 0,C 180,E1 -6460.547,E2 -6460.547} C_VEL
LIN {X 0,Y 407.302,Z 799.516,A -85,B 0,C 180,E1 -6461.76,E2 -6461.76} C_VEL
LIN {X 0,Y 406.241,Z 813.641,A -85,B 0,C 180,E1 -6463.116,E2 -6463.116} C_VEL
LIN {X 0,Y 405.175,Z 826.774,A -85,B 0,C 180,E1 -6464.689,E2 -6464.689} C_VEL
LIN {X 0,Y 404.187,Z 838.317,A -85,B 0,C 180,E1 -6466.408,E2 -6466.408} C_VEL
LIN {X 0,Y 403.278,Z 849.169,A -85,B 0,C 180,E1 -6468.414,E2 -6468.414} C_VEL
LIN {X 0,Y 402.593,Z 857.721,A -85,B 0,C 180,E1 -6470.421,E2 -6470.421} C_VEL
LIN {X 0,Y 402.074,Z 865.323,A -85,B 0,C 180,E1 -6472.713,E2 -6472.713} C_VEL
LIN {X 0,Y 401.765,Z 870.792,A -85,B 0,C 180,E1 -6475.003,E2 -6475.003} C_VEL
LIN {X 0,Y 401.665,Z 874.489,A -85,B 0,C 180,E1 -6477.289,E2 -6477.289} C_VEL
LIN {X 0,Y 401.704,Z 876.474,A -85,B 0,C 180,E1 -6479.714,E2 -6479.714} C_VEL
LIN {X 0,Y 401.884,Z 876.681,A -85,B 0,C 180,E1 -6481.996,E2 -6481.996} C_VEL
LIN {X 0,Y 402.244,Z 875.008,A -85,B 0,C 180,E1 -6484.419,E2 -6484.419} C_VEL
LIN {X 0,Y 402.789,Z 871.704,A -85,B 0,C 180,E1 -6486.7,E2 -6486.7} C_VEL
LIN {X 0,Y 403.656,Z 866.171,A -85,B 0,C 180,E1 -6489.121,E2 -6489.121} C_VEL
LIN {X 0,Y 404.678,Z 859.313,A -85,B 0,C 180,E1 -6491.255,E2 -6491.255} C_VEL
LIN {X 0,Y 405.871,Z 851.054,A -85,B 0,C 180,E1 -6493.244,E2 -6493.244} C_VEL
LIN {X 0,Y 407.223,Z 841.303,A -85,B 0,C 180,E1 -6495.085,E2 -6495.085} C_VEL
LIN {X 0,Y 408.68,Z 830.135,A -85,B 0,C 180,E1 -6496.779,E2 -6496.779} C_VEL
LIN {X 0,Y 410.23,Z 816.709,A -85,B 0,C 180,E1 -6498.399,E2 -6498.399} C_VEL
LIN {X 0,Y 411.512,Z 803.358,A -85,B 0,C 180,E1 -6499.664,E2 -6499.664} C_VEL
LIN {X 0,Y 412.629,Z 789.427,A -85,B 0,C 180,E1 -6500.718,E2 -6500.718} C_VEL
LIN {X 0,Y 413.597,Z 772.548,A -85,B 0,C 180,E1 -6501.67,E2 -6501.67} C_VEL
LIN {X 0,Y 415.527,Z 742.251,A -85,B 0,C 180,E1 -6502.933,E2 -6502.933} C_VEL
LIN {X 0,Y 427.598,Z 648.035,A -85,B 0,C 180,E1 -6506.522,E2 -6506.522} C_VEL
LIN {X 0,Y 429.332,Z 636.864,A -85,B 0,C 180,E1 -6506.934,E2 -6506.934} C_VEL
LIN {X 0,Y 434.708,Z 623.971,A -85,B 0,C 180,E1 -6507.834,E2 -6507.834} C_VEL
LIN {X 0,Y 442.309,Z 597.469,A -85,B 0,C 180,E1 -6510.873,E2 -6510.873} C_VEL
LIN {X 0,Y 450.753,Z 575.724,A -85,B 0,C 180,E1 -6513.527,E2 -6513.527} C_VEL
LIN {X 0,Y 459.461,Z 559.193,A -85,B 0,C 180,E1 -6515.676,E2 -6515.676} C_VEL
LIN {X 0,Y 462.17,Z 554.954,A -85,B 0,C 180,E1 -6516.263,E2 -6516.263} C_VEL
LIN {X 0,Y 459.132,Z 562.261,A -85,B 0,C 180,E1 -6517.766,E2 -6517.766} C_VEL
LIN {X 0,Y 458.076,Z 570.291,A -85,B 0,C 180,E1 -6519.433,E2 -6519.433} C_VEL
LIN {X 0,Y 459.347,Z 578.436,A -85,B 0,C 180,E1 -6521.099,E2 -6521.099} C_VEL
LIN {X 0,Y 462.884,Z 586.725,A -85,B 0,C 180,E1 -6522.741,E2 -6522.741} C_VEL
LIN {X 0,Y 469.09,Z 595.557,A -85,B 0,C 180,E1 -6524.434,E2 -6524.434} C_VEL
LIN {X 0,Y 475.358,Z 602.434,A -85,B 0,C 180,E1 -6525.683,E2 -6525.683} C_VEL
LIN {X 0,Y 462.53,Z 626.011,A -85,B 0,C 180,E1 -6526.22,E2 -6526.22} C_VEL
LIN {X 0,Y 453.661,Z 644.966,A -85,B 0,C 180,E1 -6526.816,E2 -6526.816} C_VEL
LIN {X 0,Y 448.627,Z 656.966,A -85,B 0,C 180,E1 -6527.262,E2 -6527.262} C_VEL
LIN {X 0,Y 440.483,Z 675.589,A -85,B 0,C 180,E1 -6527.924,E2 -6527.924} C_VEL
LIN {X 0,Y 431.178,Z 702.228,A -85,B 0,C 180,E1 -6529.09,E2 -6529.09} C_VEL
LIN {X 0,Y 428.661,Z 725.189,A -85,B 0,C 180,E1 -6529.451,E2 -6529.451} C_VEL
LIN {X 0,Y 427.08,Z 752.093,A -85,B 0,C 180,E1 -6530.119,E2 -6530.119} C_VEL
LIN {X 0,Y 424.714,Z 778.175,A -85,B 0,C 180,E1 -6531.005,E2 -6531.005} C_VEL
LIN {X 0,Y 422.36,Z 801.403,A -85,B 0,C 180,E1 -6532.054,E2 -6532.054} C_VEL
LIN {X 0,Y 419.707,Z 825.027,A -85,B 0,C 180,E1 -6533.4,E2 -6533.4} C_VEL
LIN {X 0,Y 417.009,Z 847.667,A -85,B 0,C 180,E1 -6534.976,E2 -6534.976} C_VEL
LIN {X 0,Y 414.432,Z 868.451,A -85,B 0,C 180,E1 -6536.71,E2 -6536.71} C_VEL
LIN {X 0,Y 411.819,Z 888.757,A -85,B 0,C 180,E1 -6538.717,E2 -6538.717} C_VEL
LIN {X 0,Y 409.434,Z 907.045,A -85,B 0,C 180,E1 -6540.843,E2 -6540.843} C_VEL
LIN {X 0,Y 407.247,Z 923.961,A -85,B 0,C 180,E1 -6543.143,E2 -6543.143} C_VEL
LIN {X 0,Y 405.265,Z 939.763,A -85,B 0,C 180,E1 -6545.668,E2 -6545.668} C_VEL
LIN {X 0,Y 403.511,Z 954.584,A -85,B 0,C 180,E1 -6548.486,E2 -6548.486} C_VEL
LIN {X 0,Y 402.199,Z 966.886,A -85,B 0,C 180,E1 -6551.295,E2 -6551.295} C_VEL
LIN {X 0,Y 401.287,Z 977.023,A -85,B 0,C 180,E1 -6554.104,E2 -6554.104} C_VEL
LIN {X 0,Y 400.696,Z 985.186,A -85,B 0,C 180,E1 -6556.875,E2 -6556.875} C_VEL
LIN {X 0,Y 400.33,Z 991.963,A -85,B 0,C 180,E1 -6559.785,E2 -6559.785} C_VEL
LIN {X 0,Y 400.172,Z 996.702,A -85,B 0,C 180,E1 -6562.534,E2 -6562.534} C_VEL
LIN {X 0,Y 400.132,Z 1000.131,A -85,B 0,C 180,E1 -6565.413,E2 -6565.413} C_VEL
LIN {X 0,Y 400.119,Z 1001.94,A -85,B 0,C 180,E1 -6568.424,E2 -6568.424} C_VEL
LIN {X 0,Y 400.121,Z 1002.139,A -85,B 0,C 180,E1 -6571.145,E2 -6571.145} C_VEL
LIN {X 0,Y 400.116,Z 1000.668,A -85,B 0,C 180,E1 -6574.155,E2 -6574.155} C_VEL
LIN {X 0,Y 400.123,Z 997.697,A -85,B 0,C 180,E1 -6577.033,E2 -6577.033} C_VEL
LIN {X 0,Y 400.257,Z 992.851,A -85,B 0,C 180,E1 -6580.07,E2 -6580.07} C_VEL
LIN {X 0,Y 400.601,Z 986.485,A -85,B 0,C 180,E1 -6582.981,E2 -6582.981} C_VEL
LIN {X 0,Y 401.224,Z 978.352,A -85,B 0,C 180,E1 -6585.909,E2 -6585.909} C_VEL
LIN {X 0,Y 402.216,Z 968.272,A -85,B 0,C 180,E1 -6588.854,E2 -6588.854} C_VEL
LIN {X 0,Y 403.684,Z 956.016,A -85,B 0,C 180,E1 -6591.809,E2 -6591.809} C_VEL
LIN {X 0,Y 405.585,Z 942.073,A -85,B 0,C 180,E1 -6594.621,E2 -6594.621} C_VEL
LIN {X 0,Y 407.976,Z 925.955,A -85,B 0,C 180,E1 -6597.356,E2 -6597.356} C_VEL
LIN {X 0,Y 410.682,Z 908.433,A -85,B 0,C 180,E1 -6599.86,E2 -6599.86} C_VEL
LIN {X 0,Y 413.529,Z 890.292,A -85,B 0,C 180,E1 -6602.054,E2 -6602.054} C_VEL
LIN {X 0,Y 416.389,Z 871.553,A -85,B 0,C 180,E1 -6603.967,E2 -6603.967} C_VEL
LIN {X 0,Y 419.409,Z 850.942,A -85,B 0,C 180,E1 -6605.737,E2 -6605.737} C_VEL
LIN {X 0,Y 422.158,Z 831.272,A -85,B 0,C 180,E1 -6607.153,E2 -6607.153} C_VEL
LIN {X 0,Y 424.775,Z 810.103,A -85,B 0,C 180,E1 -6608.388,E2 -6608.388} C_VEL
LIN {X 0,Y 427.244,Z 787.64,A -85,B 0,C 180,E1 -6609.427,E2 -6609.427} C_VEL
LIN {X 0,Y 429.266,Z 765.99,A -85,B 0,C 180,E1 -6610.191,E2 -6610.191} C_VEL
LIN {X 0,Y 430.692,Z 743.181,A -85,B 0,C 180,E1 -6610.757,E2 -6610.757} C_VEL
LIN {X 0,Y 431.993,Z 716.952,A -85,B 0,C 180,E1 -6611.25,E2 -6611.25} C_VEL
LIN {X 0,Y 432.761,Z 711.207,A -85,B 0,C 180,E1 -6611.359,E2 -6611.359} C_VEL
LIN {X 0,Y 438.631,Z 694.093,A -85,B 0,C 180,E1 -6612.168,E2 -6612.168} C_VEL
LIN {X 0,Y 445.798,Z 675.156,A -85,B 0,C 180,E1 -6612.986,E2 -6612.986} C_VEL
LIN {X 0,Y 455.231,Z 654.36,A -85,B 0,C 180,E1 -6613.721,E2 -6613.721} C_VEL
LIN {X 0,Y 463.452,Z 636.131,A -85,B 0,C 180,E1 -6614.347,E2 -6614.347} C_VEL
LIN {X 0,Y 474.659,Z 614.881,A -85,B 0,C 180,E1 -6614.883,E2 -6614.883} C_VEL
LIN {X 0,Y 479.793,Z 605.743,A -85,B 0,C 180,E1 -6615.074,E2 -6615.074} C_VEL
LIN {X 0,Y 470.427,Z 595.366,A -85,B 0,C 180,E1 -6616.813,E2 -6616.813} C_VEL
LIN {X 0,Y 462.583,Z 583.582,A -85,B 0,C 180,E1 -6618.593,E2 -6618.593} C_VEL
LIN {X 0,Y 456.034,Z 569.418,A -85,B 0,C 180,E1 -6620.519,E2 -6620.519} C_VEL
LIN {X 0,Y 451.608,Z 554.576,A -85,B 0,C 180,E1 -6622.334,E2 -6622.334} C_VEL
LIN {X 0,Y 448.933,Z 538.154,A -85,B 0,C 180,E1 -6624.144,E2 -6624.144} C_VEL
LIN {X 0,Y 448.083,Z 519.361,A -85,B 0,C 180,E1 -6626.016,E2 -6626.016} C_VEL
LIN {X 0,Y 449.117,Z 499.476,A -85,B 0,C 180,E1 -6627.777,E2 -6627.777} C_VEL
LIN {X 0,Y 452.64,Z 471.712,A -85,B 0,C 180,E1 -6630.015,E2 -6630.015} C_VEL
LIN {X 0,Y 442.979,Z 453.559,A -85,B 0,C 180,E1 -6633.455,E2 -6633.455} C_VEL
LIN {X 0,Y 433.188,Z 435.772,A -85,B 0,C 180,E1 -6637.185,E2 -6637.185} C_VEL
LIN {X 0,Y 425.082,Z 421.514,A -85,B 0,C 180,E1 -6640.488,E2 -6640.488} C_VEL
LIN {X 0,Y 418.456,Z 410.277,A -85,B 0,C 180,E1 -6643.338,E2 -6643.338} C_VEL
LIN {X 0,Y 415.83,Z 405.745,A -85,B 0,C 180,E1 -6644.521,E2 -6644.521} C_VEL
LIN {X 0,Y 412.981,Z 400.882,A -85,B 0,C 180,E1 -6645.846,E2 -6645.846} C_VEL
LIN {X 0,Y 410.096,Z 395.959,A -85,B 0,C 180,E1 -6647.223,E2 -6647.223} C_VEL
LIN {X 0,Y 407.961,Z 392.391,A -85,B 0,C 180,E1 -6648.263,E2 -6648.263} C_VEL
LIN {X 0,Y 407.176,Z 390.93,A -85,B 0,C 180,E1 -6648.671,E2 -6648.671} C_VEL
LIN {X 0,Y 404.958,Z 387.434,A -85,B 0,C 180,E1 -6649.76,E2 -6649.76} C_VEL
LIN {X 0,Y 404.283,Z 385.85,A -85,B 0,C 180,E1 -6650.175,E2 -6650.175} C_VEL
LIN {X 0,Y 401.961,Z 382.591,A -85,B 0,C 180,E1 -6651.273,E2 -6651.273} C_VEL
LIN {X 0,Y 401.501,Z 380.721,A -85,B 0,C 180,E1 -6651.696,E2 -6651.696} C_VEL
LIN {X 0,Y 401.46,Z 380.73,A -85,B 0,C 180,E1 -6655.572,E2 -6655.572} C_VEL
LIN {X 0,Y 401.505,Z 380.729,A -85,B 0,C 180,E1 -6659.572,E2 -6659.572} C_VEL
LIN {X 0,Y 401.472,Z 380.729,A -85,B 0,C 180,E1 -6663.427,E2 -6663.427} C_VEL
LIN {X 0,Y 401.511,Z 380.724,A -85,B 0,C 180,E1 -6667.297,E2 -6667.297} C_VEL
LIN {X 0,Y 401.493,Z 380.728,A -85,B 0,C 180,E1 -6671.347,E2 -6671.347} C_VEL
LIN {X 0,Y 401.491,Z 380.72,A -85,B 0,C 180,E1 -6675.159,E2 -6675.159} C_VEL
LIN {X 0,Y 401.486,Z 380.724,A -85,B 0,C 180,E1 -6679.192,E2 -6679.192} C_VEL
LIN {X 0,Y 401.484,Z 380.723,A -85,B 0,C 180,E1 -6683.017,E2 -6683.017} C_VEL
LIN {X 0,Y 401.477,Z 380.714,A -85,B 0,C 180,E1 -6687.114,E2 -6687.114} C_VEL
LIN {X 0,Y 401.487,Z 380.714,A -85,B 0,C 180,E1 -6690.866,E2 -6690.866} C_VEL
LIN {X 0,Y 401.475,Z 380.699,A -85,B 0,C 180,E1 -6694.979,E2 -6694.979} C_VEL
LIN {X 0,Y 401.488,Z 380.717,A -85,B 0,C 180,E1 -6698.872,E2 -6698.872} C_VEL
LIN {X 0,Y 401.481,Z 380.692,A -85,B 0,C 180,E1 -6702.931,E2 -6702.931} C_VEL
LIN {X 0,Y 401.518,Z 380.831,A -85,B 0,C 180,E1 -6704.697,E2 -6704.697} C_VEL
LIN {X 0,Y 402.851,Z 384.279,A -85,B 0,C 180,E1 -6705.181,E2 -6705.181} C_VEL
LIN {X 0,Y 403.885,Z 386.098,A -85,B 0,C 180,E1 -6705.478,E2 -6705.478} C_VEL
LIN {X 0,Y 411.467,Z 401.768,A -85,B 0,C 180,E1 -6707.83,E2 -6707.83} C_VEL
LIN {X 0,Y 418.658,Z 418.472,A -85,B 0,C 180,E1 -6710.17,E2 -6710.17} C_VEL
LIN {X 0,Y 424.839,Z 435.417,A -85,B 0,C 180,E1 -6712.358,E2 -6712.358} C_VEL
LIN {X 0,Y 422.794,Z 477.453,A -85,B 0,C 180,E1 -6715.658,E2 -6715.658} C_VEL
LIN {X 0,Y 422.417,Z 495.474,A -85,B 0,C 180,E1 -6716.937,E2 -6716.937} C_VEL
LIN {X 0,Y 423.344,Z 503.528,A -85,B 0,C 180,E1 -6717.183,E2 -6717.183} C_VEL
LIN {X 0,Y 418.743,Z 701.738,A -85,B 0,C 180,E1 -6720.737,E2 -6720.737} C_VEL
LIN {X 0,Y 418.182,Z 721.023,A -85,B 0,C 180,E1 -6721.324,E2 -6721.324} C_VEL
LIN {X 0,Y 417.219,Z 739.289,A -85,B 0,C 180,E1 -6722.14,E2 -6722.14} C_VEL
LIN {X 0,Y 416.316,Z 751.71,A -85,B 0,C 180,E1 -6722.851,E2 -6722.851} C_VEL
LIN {X 0,Y 414.808,Z 758.954,A -85,B 0,C 180,E1 -6723.255,E2 -6723.255} C_VEL
LIN {X 0,Y 408.125,Z 775.573,A -85,B 0,C 180,E1 -6724.138,E2 -6724.138} C_VEL
LIN {X 0,Y 406.312,Z 782.007,A -85,B 0,C 180,E1 -6724.641,E2 -6724.641} C_VEL
LIN {X 0,Y 406.191,Z 782.909,A -85,B 0,C 180,E1 -6724.724,E2 -6724.724} C_VEL
LIN {X 0,Y 404.183,Z 798.346,A -85,B 0,C 180,E1 -6726.375,E2 -6726.375} C_VEL
LIN {X 0,Y 402.097,Z 812.65,A -85,B 0,C 180,E1 -6728.254,E2 -6728.254} C_VEL
LIN {X 0,Y 400.137,Z 825.358,A -85,B 0,C 180,E1 -6730.286,E2 -6730.286} C_VEL
LIN {X 0,Y 398.329,Z 836.606,A -85,B 0,C 180,E1 -6732.47,E2 -6732.47} C_VEL
LIN {X 0,Y 396.755,Z 846.555,A -85,B 0,C 180,E1 -6734.84,E2 -6734.84} C_VEL
LIN {X 0,Y 395.453,Z 855.175,A -85,B 0,C 180,E1 -6737.413,E2 -6737.413} C_VEL
LIN {X 0,Y 394.481,Z 862.086,A -85,B 0,C 180,E1 -6740.076,E2 -6740.076} C_VEL
LIN {X 0,Y 393.841,Z 867.367,A -85,B 0,C 180,E1 -6742.854,E2 -6742.854} C_VEL
LIN {X 0,Y 393.486,Z 870.845,A -85,B 0,C 180,E1 -6745.628,E2 -6745.628} C_VEL
LIN {X 0,Y 393.312,Z 872.64,A -85,B 0,C 180,E1 -6748.398,E2 -6748.398} C_VEL
LIN {X 0,Y 393.293,Z 872.803,A -85,B 0,C 180,E1 -6751.166,E2 -6751.166} C_VEL
LIN {X 0,Y 393.438,Z 871.338,A -85,B 0,C 180,E1 -6753.935,E2 -6753.935} C_VEL
LIN {X 0,Y 393.762,Z 868.208,A -85,B 0,C 180,E1 -6756.708,E2 -6756.708} C_VEL
LIN {X 0,Y 394.339,Z 863.283,A -85,B 0,C 180,E1 -6759.487,E2 -6759.487} C_VEL
LIN {X 0,Y 395.224,Z 856.82,A -85,B 0,C 180,E1 -6762.122,E2 -6762.122} C_VEL
LIN {X 0,Y 396.405,Z 848.931,A -85,B 0,C 180,E1 -6764.61,E2 -6764.61} C_VEL
LIN {X 0,Y 397.852,Z 839.669,A -85,B 0,C 180,E1 -6766.95,E2 -6766.95} C_VEL
LIN {X 0,Y 399.556,Z 829.064,A -85,B 0,C 180,E1 -6769.137,E2 -6769.137} C_VEL
LIN {X 0,Y 401.43,Z 817.108,A -85,B 0,C 180,E1 -6771.172,E2 -6771.172} C_VEL
LIN {X 0,Y 403.422,Z 803.721,A -85,B 0,C 180,E1 -6773.054,E2 -6773.054} C_VEL
LIN {X 0,Y 405.384,Z 789.428,A -85,B 0,C 180,E1 -6774.713,E2 -6774.713} C_VEL
LIN {X 0,Y 407.274,Z 773.49,A -85,B 0,C 180,E1 -6776.226,E2 -6776.226} C_VEL
LIN {X 0,Y 408.886,Z 757.618,A -85,B 0,C 180,E1 -6777.441,E2 -6777.441} C_VEL
LIN {X 0,Y 410.276,Z 740.366,A -85,B 0,C 180,E1 -6778.48,E2 -6778.48} C_VEL
LIN {X 0,Y 411.293,Z 721.84,A -85,B 0,C 180,E1 -6779.316,E2 -6779.316} C_VEL
LIN {X 0,Y 411.869,Z 702.602,A -85,B 0,C 180,E1 -6779.906,E2 -6779.906} C_VEL
LIN {X 0,Y 416.595,Z 502.241,A -85,B 0,C 180,E1 -6783.567,E2 -6783.567} C_VEL
LIN {X 0,Y 415.734,Z 495.277,A -85,B 0,C 180,E1 -6783.833,E2 -6783.833} C_VEL
LIN {X 0,Y 417.013,Z 461.123,A -85,B 0,C 180,E1 -6786.401,E2 -6786.401} C_VEL
LIN {X 0,Y 418.119,Z 438.179,A -85,B 0,C 180,E1 -6788.27,E2 -6788.27} C_VEL
LIN {X 0,Y 410.879,Z 419.004,A -85,B 0,C 180,E1 -6790.816,E2 -6790.816} C_VEL
LIN {X 0,Y 404.29,Z 404.001,A -85,B 0,C 180,E1 -6792.993,E2 -6792.993} C_VEL
LIN {X 0,Y 403.904,Z 403.887,A -85,B 0,C 180,E1 -6793.098,E2 -6793.098} C_VEL
LIN {X 0,Y 410.759,Z 419.298,A -85,B 0,C 180,E1 -6795.897,E2 -6795.897} C_VEL
LIN {X 0,Y 418.019,Z 437.438,A -85,B 0,C 180,E1 -6798.891,E2 -6798.891} C_VEL
LIN {X 0,Y 421.064,Z 445.475,A -85,B 0,C 180,E1 -6800.123,E2 -6800.123} C_VEL
LIN {X 0,Y 416.723,Z 486.998,A -85,B 0,C 180,E1 -6804.081,E2 -6804.081} C_VEL
LIN {X 0,Y 412.479,Z 531.673,A -85,B 0,C 180,E1 -6808.263,E2 -6808.263} C_VEL
LIN {X 0,Y 408.621,Z 577.055,A -85,B 0,C 180,E1 -6812.453,E2 -6812.453} C_VEL
LIN {X 0,Y 406.615,Z 604.568,A -85,B 0,C 180,E1 -6814.936,E2 -6814.936} C_VEL
LIN {X 0,Y 407.354,Z 613.72,A -85,B 0,C 180,E1 -6815.236,E2 -6815.236} C_VEL
LIN {X 0,Y 402.143,Z 750.614,A -85,B 0,C 180,E1 -6818.598,E2 -6818.598} C_VEL
LIN {X 0,Y 401.605,Z 767.024,A -85,B 0,C 180,E1 -6819.241,E2 -6819.241} C_VEL
LIN {X 0,Y 400.78,Z 783.651,A -85,B 0,C 180,E1 -6820.166,E2 -6820.166} C_VEL
LIN {X 0,Y 399.774,Z 799.151,A -85,B 0,C 180,E1 -6821.328,E2 -6821.328} C_VEL
LIN {X 0,Y 398.665,Z 813.638,A -85,B 0,C 180,E1 -6822.71,E2 -6822.71} C_VEL
LIN {X 0,Y 397.487,Z 827.517,A -85,B 0,C 180,E1 -6824.386,E2 -6824.386} C_VEL
LIN {X 0,Y 396.449,Z 839.182,A -85,B 0,C 180,E1 -6826.137,E2 -6826.137} C_VEL
LIN {X 0,Y 395.488,Z 850.11,A -85,B 0,C 180,E1 -6828.183,E2 -6828.183} C_VEL
LIN {X 0,Y 394.765,Z 858.764,A -85,B 0,C 180,E1 -6830.229,E2 -6830.229} C_VEL
LIN {X 0,Y 394.211,Z 866.441,A -85,B 0,C 180,E1 -6832.567,E2 -6832.567} C_VEL
LIN {X 0,Y 393.883,Z 871.998,A -85,B 0,C 180,E1 -6834.902,E2 -6834.902} C_VEL
LIN {X 0,Y 393.778,Z 875.78,A -85,B 0,C 180,E1 -6837.234,E2 -6837.234} C_VEL
LIN {X 0,Y 393.812,Z 877.784,A -85,B 0,C 180,E1 -6839.563,E2 -6839.563} C_VEL
LIN {X 0,Y 394.023,Z 878.145,A -85,B 0,C 180,E1 -6842.035,E2 -6842.035} C_VEL
LIN {X 0,Y 394.418,Z 876.559,A -85,B 0,C 180,E1 -6844.507,E2 -6844.507} C_VEL
LIN {X 0,Y 395.016,Z 873.365,A -85,B 0,C 180,E1 -6846.832,E2 -6846.832} C_VEL
LIN {X 0,Y 395.95,Z 867.92,A -85,B 0,C 180,E1 -6849.3,E2 -6849.3} C_VEL
LIN {X 0,Y 397.054,Z 861.189,A -85,B 0,C 180,E1 -6851.474,E2 -6851.474} C_VEL
LIN {X 0,Y 398.339,Z 853.079,A -85,B 0,C 180,E1 -6853.499,E2 -6853.499} C_VEL
LIN {X 0,Y 399.779,Z 843.477,A -85,B 0,C 180,E1 -6855.373,E2 -6855.373} C_VEL
LIN {X 0,Y 401.343,Z 832.568,A -85,B 0,C 180,E1 -6857.095,E2 -6857.095} C_VEL
LIN {X 0,Y 402.987,Z 819.396,A -85,B 0,C 180,E1 -6858.741,E2 -6858.741} C_VEL
LIN {X 0,Y 404.366,Z 806.692,A -85,B 0,C 180,E1 -6860.013,E2 -6860.013} C_VEL
LIN {X 0,Y 405.659,Z 792.158,A -85,B 0,C 180,E1 -6861.167,E2 -6861.167} C_VEL
LIN {X 0,Y 406.783,Z 775.469,A -85,B 0,C 180,E1 -6862.166,E2 -6862.166} C_VEL
LIN {X 0,Y 408.877,Z 746.231,A -85,B 0,C 180,E1 -6863.471,E2 -6863.471} C_VEL
LIN {X 0,Y 420.894,Z 660.363,A -85,B 0,C 180,E1 -6866.935,E2 -6866.935} C_VEL
LIN {X 0,Y 423.996,Z 640.088,A -85,B 0,C 180,E1 -6867.681,E2 -6867.681} C_VEL
LIN {X 0,Y 429.923,Z 626.482,A -85,B 0,C 180,E1 -6868.625,E2 -6868.625} C_VEL
LIN {X 0,Y 437.779,Z 601.772,A -85,B 0,C 180,E1 -6871.535,E2 -6871.535} C_VEL
LIN {X 0,Y 446.833,Z 580.704,A -85,B 0,C 180,E1 -6874.17,E2 -6874.17} C_VEL
LIN {X 0,Y 455.589,Z 565.548,A -85,B 0,C 180,E1 -6876.182,E2 -6876.182} C_VEL
LIN {X 0,Y 456.66,Z 563.971,A -85,B 0,C 180,E1 -6876.434,E2 -6876.434} C_VEL
LIN {X 0,Y 453.893,Z 571.877,A -85,B 0,C 180,E1 -6878.147,E2 -6878.147} C_VEL
LIN {X 0,Y 453.561,Z 579.99,A -85,B 0,C 180,E1 -6879.903,E2 -6879.903} C_VEL
LIN {X 0,Y 455.703,Z 588.386,A -85,B 0,C 180,E1 -6881.667,E2 -6881.667} C_VEL
LIN {X 0,Y 460.205,Z 596.673,A -85,B 0,C 180,E1 -6883.357,E2 -6883.357} C_VEL
LIN {X 0,Y 467.117,Z 605.2,A -85,B 0,C 180,E1 -6885.026,E2 -6885.026} C_VEL
LIN {X 0,Y 467.268,Z 605.625,A -85,B 0,C 180,E1 -6885.078,E2 -6885.078} C_VEL
LIN {X 0,Y 455.257,Z 628.233,A -85,B 0,C 180,E1 -6885.612,E2 -6885.612} C_VEL
LIN {X 0,Y 446.626,Z 647.075,A -85,B 0,C 180,E1 -6886.23,E2 -6886.23} C_VEL
LIN {X 0,Y 442.336,Z 657.035,A -85,B 0,C 180,E1 -6886.593,E2 -6886.593} C_VEL
LIN {X 0,Y 434.089,Z 675.959,A -85,B 0,C 180,E1 -6887.277,E2 -6887.277} C_VEL
LIN {X 0,Y 425.457,Z 700.291,A -85,B 0,C 180,E1 -6888.345,E2 -6888.345} C_VEL
LIN {X 0,Y 422.55,Z 725.211,A -85,B 0,C 180,E1 -6888.753,E2 -6888.753} C_VEL
LIN {X 0,Y 420.729,Z 751.624,A -85,B 0,C 180,E1 -6889.45,E2 -6889.45} C_VEL
LIN {X 0,Y 418.064,Z 778.282,A -85,B 0,C 180,E1 -6890.397,E2 -6890.397} C_VEL
LIN {X 0,Y 415.314,Z 802.608,A -85,B 0,C 180,E1 -6891.557,E2 -6891.557} C_VEL
LIN {X 0,Y 412.457,Z 826.15,A -85,B 0,C 180,E1 -6892.957,E2 -6892.957} C_VEL
LIN {X 0,Y 409.604,Z 848.346,A -85,B 0,C 180,E1 -6894.567,E2 -6894.567} C_VEL
LIN {X 0,Y 406.677,Z 870.381,A -85,B 0,C 180,E1 -6896.49,E2 -6896.49} C_VEL
LIN {X 0,Y 403.897,Z 890.762,A -85,B 0,C 180,E1 -6898.593,E2 -6898.593} C_VEL
LIN {X 0,Y 401.285,Z 909.871,A -85,B 0,C 180,E1 -6900.93,E2 -6900.93} C_VEL
LIN {X 0,Y 398.899,Z 927.561,A -85,B 0,C 180,E1 -6903.486,E2 -6903.486} C_VEL
LIN {X 0,Y 396.917,Z 942.993,A -85,B 0,C 180,E1 -6906.122,E2 -6906.122} C_VEL
LIN {X 0,Y 395.236,Z 957.061,A -85,B 0,C 180,E1 -6908.984,E2 -6908.984} C_VEL
LIN {X 0,Y 393.955,Z 969.198,A -85,B 0,C 180,E1 -6911.962,E2 -6911.962} C_VEL
LIN {X 0,Y 393.117,Z 978.716,A -85,B 0,C 180,E1 -6914.812,E2 -6914.812} C_VEL
LIN {X 0,Y 392.611,Z 986.387,A -85,B 0,C 180,E1 -6917.647,E2 -6917.647} C_VEL
LIN {X 0,Y 392.316,Z 992.878,A -85,B 0,C 180,E1 -6920.76,E2 -6920.76} C_VEL
LIN {X 0,Y 392.237,Z 997.224,A -85,B 0,C 180,E1 -6923.707,E2 -6923.707} C_VEL
LIN {X 0,Y 392.203,Z 999.845,A -85,B 0,C 180,E1 -6926.492,E2 -6926.492} C_VEL
LIN {X 0,Y 392.191,Z 1001.008,A -85,B 0,C 180,E1 -6929.269,E2 -6929.269} C_VEL
LIN {X 0,Y 392.188,Z 1000.736,A -85,B 0,C 180,E1 -6932.191,E2 -6932.191} C_VEL
LIN {X 0,Y 392.162,Z 998.831,A -85,B 0,C 180,E1 -6935.119,E2 -6935.119} C_VEL
LIN {X 0,Y 392.208,Z 995.392,A -85,B 0,C 180,E1 -6938.06,E2 -6938.06} C_VEL
LIN {X 0,Y 392.402,Z 989.917,A -85,B 0,C 180,E1 -6941.19,E2 -6941.19} C_VEL
LIN {X 0,Y 392.813,Z 983.043,A -85,B 0,C 180,E1 -6944.143,E2 -6944.143} C_VEL
LIN {X 0,Y 393.578,Z 974.293,A -85,B 0,C 180,E1 -6947.139,E2 -6947.139} C_VEL
LIN {X 0,Y 394.779,Z 963.518,A -85,B 0,C 180,E1 -6950.148,E2 -6950.148} C_VEL
LIN {X 0,Y 396.496,Z 950.463,A -85,B 0,C 180,E1 -6953.165,E2 -6953.165} C_VEL
LIN {X 0,Y 398.69,Z 935.608,A -85,B 0,C 180,E1 -6956.032,E2 -6956.032} C_VEL
LIN {X 0,Y 401.333,Z 919.008,A -85,B 0,C 180,E1 -6958.724,E2 -6958.724} C_VEL
LIN {X 0,Y 404.246,Z 901.266,A -85,B 0,C 180,E1 -6961.153,E2 -6961.153} C_VEL
LIN {X 0,Y 407.107,Z 883.453,A -85,B 0,C 180,E1 -6963.208,E2 -6963.208} C_VEL
LIN {X 0,Y 410.2,Z 864.055,A -85,B 0,C 180,E1 -6965.117,E2 -6965.117} C_VEL
LIN {X 0,Y 413.129,Z 844.78,A -85,B 0,C 180,E1 -6966.711,E2 -6966.711} C_VEL
LIN {X 0,Y 415.929,Z 824.729,A -85,B 0,C 180,E1 -6968.086,E2 -6968.086} C_VEL
LIN {X 0,Y 418.624,Z 803.734,A -85,B 0,C 180,E1 -6969.267,E2 -6969.267} C_VEL
LIN {X 0,Y 420.991,Z 781.993,A -85,B 0,C 180,E1 -6970.224,E2 -6970.224} C_VEL
LIN {X 0,Y 423.033,Z 759.468,A -85,B 0,C 180,E1 -6970.958,E2 -6970.958} C_VEL
LIN {X 0,Y 424.438,Z 734.637,A -85,B 0,C 180,E1 -6971.539,E2 -6971.539} C_VEL
LIN {X 0,Y 425.636,Z 715.076,A -85,B 0,C 180,E1 -6971.892,E2 -6971.892} C_VEL
LIN {X 0,Y 426.172,Z 710.857,A -85,B 0,C 180,E1 -6971.962,E2 -6971.962} C_VEL
LIN {X 0,Y 432.464,Z 692.935,A -85,B 0,C 180,E1 -6972.822,E2 -6972.822} C_VEL
LIN {X 0,Y 439.699,Z 674.077,A -85,B 0,C 180,E1 -6973.641,E2 -6973.641} C_VEL
LIN {X 0,Y 449.05,Z 653.635,A -85,B 0,C 180,E1 -6974.359,E2 -6974.359} C_VEL
LIN {X 0,Y 457.453,Z 635.116,A -85,B 0,C 180,E1 -6974.997,E2 -6974.997} C_VEL
LIN {X 0,Y 469.147,Z 613.178,A -85,B 0,C 180,E1 -6975.558,E2 -6975.558} C_VEL
LIN {X 0,Y 471.565,Z 608.787,A -85,B 0,C 180,E1 -6975.657,E2 -6975.657} C_VEL
LIN {X 0,Y 461.968,Z 597.091,A -85,B 0,C 180,E1 -6977.564,E2 -6977.564} C_VEL
LIN {X 0,Y 454.801,Z 585.094,A -85,B 0,C 180,E1 -6979.329,E2 -6979.329} C_VEL
LIN {X 0,Y 448.81,Z 570.775,A -85,B 0,C 180,E1 -6981.244,E2 -6981.244} C_VEL
LIN {X 0,Y 444.871,Z 555.927,A -85,B 0,C 180,E1 -6983.044,E2 -6983.044} C_VEL
LIN {X 0,Y 442.6,Z 539.416,A -85,B 0,C 180,E1 -6984.863,E2 -6984.863} C_VEL
LIN {X 0,Y 442.011,Z 520.531,A -85,B 0,C 180,E1 -6986.733,E2 -6986.733} C_VEL
LIN {X 0,Y 443.484,Z 499.31,A -85,B 0,C 180,E1 -6988.614,E2 -6988.614} C_VEL
LIN {X 0,Y 446.602,Z 476.067,A -85,B 0,C 180,E1 -6990.493,E2 -6990.493} C_VEL
LIN {X 0,Y 437.426,Z 458.751,A -85,B 0,C 180,E1 -6993.823,E2 -6993.823} C_VEL
LIN {X 0,Y 427.964,Z 441.477,A -85,B 0,C 180,E1 -6997.471,E2 -6997.471} C_VEL
LIN {X 0,Y 419.862,Z 427.215,A -85,B 0,C 180,E1 -7000.815,E2 -7000.815} C_VEL
LIN {X 0,Y 413.212,Z 415.868,A -85,B 0,C 180,E1 -7003.699,E2 -7003.699} C_VEL
LIN {X 0,Y 410.631,Z 411.384,A -85,B 0,C 180,E1 -7004.898,E2 -7004.898} C_VEL
LIN {X 0,Y 408.051,Z 406.943,A -85,B 0,C 180,E1 -7006.106,E2 -7006.106} C_VEL
LIN {X 0,Y 405.273,Z 402.163,A -85,B 0,C 180,E1 -7007.461,E2 -7007.461} C_VEL
LIN {X 0,Y 402.217,Z 397.008,A -85,B 0,C 180,E1 -7008.965,E2 -7008.965} C_VEL
LIN {X 0,Y 400.044,Z 393.362,A -85,B 0,C 180,E1 -7010.07,E2 -7010.07} C_VEL
LIN {X 0,Y 399.267,Z 391.934,A -85,B 0,C 180,E1 -7010.487,E2 -7010.487} C_VEL
LIN {X 0,Y 397.083,Z 388.5,A -85,B 0,C 180,E1 -7011.603,E2 -7011.603} C_VEL
LIN {X 0,Y 396.445,Z 386.925,A -85,B 0,C 180,E1 -7012.027,E2 -7012.027} C_VEL
LIN {X 0,Y 394.117,Z 383.786,A -85,B 0,C 180,E1 -7013.152,E2 -7013.152} C_VEL
LIN {X 0,Y 393.537,Z 381.713,A -85,B 0,C 180,E1 -7013.728,E2 -7013.728} C_VEL
LIN {X 0,Y 393.55,Z 381.715,A -85,B 0,C 180,E1 -7017.962,E2 -7017.962} C_VEL
LIN {X 0,Y 393.535,Z 381.723,A -85,B 0,C 180,E1 -7021.748,E2 -7021.748} C_VEL
LIN {X 0,Y 393.554,Z 381.715,A -85,B 0,C 180,E1 -7025.979,E2 -7025.979} C_VEL
LIN {X 0,Y 393.537,Z 381.714,A -85,B 0,C 180,E1 -7029.801,E2 -7029.801} C_VEL
LIN {X 0,Y 393.56,Z 381.713,A -85,B 0,C 180,E1 -7033.817,E2 -7033.817} C_VEL
LIN {X 0,Y 393.545,Z 381.709,A -85,B 0,C 180,E1 -7037.751,E2 -7037.751} C_VEL
LIN {X 0,Y 393.57,Z 381.709,A -85,B 0,C 180,E1 -7041.772,E2 -7041.772} C_VEL
LIN {X 0,Y 393.546,Z 381.713,A -85,B 0,C 180,E1 -7045.751,E2 -7045.751} C_VEL
LIN {X 0,Y 393.562,Z 381.712,A -85,B 0,C 180,E1 -7049.674,E2 -7049.674} C_VEL
LIN {X 0,Y 393.539,Z 381.714,A -85,B 0,C 180,E1 -7053.633,E2 -7053.633} C_VEL
LIN {X 0,Y 393.547,Z 381.673,A -85,B 0,C 180,E1 -7057.572,E2 -7057.572} C_VEL
LIN {X 0,Y 393.535,Z 381.681,A -85,B 0,C 180,E1 -7061.734,E2 -7061.734} C_VEL
LIN {X 0,Y 393.561,Z 381.721,A -85,B 0,C 180,E1 -7063.66,E2 -7063.66} C_VEL
LIN {X 0,Y 394.815,Z 385.103,A -85,B 0,C 180,E1 -7064.142,E2 -7064.142} C_VEL
LIN {X 0,Y 396.004,Z 386.986,A -85,B 0,C 180,E1 -7064.48,E2 -7064.48} C_VEL
LIN {X 0,Y 403.944,Z 403.153,A -85,B 0,C 180,E1 -7067.007,E2 -7067.007} C_VEL
LIN {X 0,Y 411.089,Z 419.474,A -85,B 0,C 180,E1 -7069.364,E2 -7069.364} C_VEL
LIN {X 0,Y 418.199,Z 438.589,A -85,B 0,C 180,E1 -7071.894,E2 -7071.894} C_VEL
LIN {X 0,Y 416.154,Z 479.607,A -85,B 0,C 180,E1 -7075.123,E2 -7075.123} C_VEL
LIN {X 0,Y 415.782,Z 496.727,A -85,B 0,C 180,E1 -7076.342,E2 -7076.342} C_VEL
LIN {X 0,Y 416.681,Z 504.814,A -85,B 0,C 180,E1 -7076.593,E2 -7076.593} C_VEL
LIN {X 0,Y 411.841,Z 702.724,A -85,B 0,C 180,E1 -7080.193,E2 -7080.193} C_VEL
LIN {X 0,Y 411.261,Z 722.021,A -85,B 0,C 180,E1 -7080.787,E2 -7080.787} C_VEL
LIN {X 0,Y 410.325,Z 739.261,A -85,B 0,C 180,E1 -7081.559,E2 -7081.559} C_VEL
LIN {X 0,Y 408.893,Z 757.257,A -85,B 0,C 180,E1 -7082.632,E2 -7082.632} C_VEL
LIN {X 0,Y 407.252,Z 773.478,A -85,B 0,C 180,E1 -7083.87,E2 -7083.87} C_VEL
